C07268=1082.285,311.899,-88.847,175.955,25.912,154.344
C07269=1082.279,311.650,-88.815,175.952,25.909,154.344
C07270=1082.273,311.403,-88.784,175.949,25.904,154.343
C07271=1082.267,311.155,-88.752,175.946,25.900,154.343
C07272=1082.262,310.908,-88.720,175.943,25.896,154.342
C07273=1082.256,310.659,-88.688,175.941,25.892,154.341
C07274=1082.249,310.411,-88.657,175.937,25.888,154.341
C07275=1082.244,310.164,-88.625,175.935,25.884,154.340
C07276=1082.238,309.916,-88.593,175.931,25.880,154.340
C07277=1082.231,309.668,-88.562,175.928,25.876,154.339
C07278=1082.226,309.420,-88.531,175.925,25.872,154.339
C07279=1082.220,309.172,-88.499,175.922,25.868,154.338
C07280=1082.214,308.924,-88.467,175.919,25.864,154.338
C07281=1082.208,308.676,-88.435,175.916,25.860,154.337
C07282=1082.202,308.429,-88.404,175.913,25.856,154.336
C07283=1082.196,308.180,-88.372,175.911,25.852,154.336
C07284=1082.190,307.932,-88.341,175.908,25.848,154.335
C07285=1082.185,307.684,-88.309,175.905,25.844,154.335
C07286=1082.179,307.437,-88.278,175.902,25.840,154.334
C07287=1082.172,307.189,-88.246,175.899,25.836,154.334
C07288=1082.167,306.941,-88.215,175.896,25.832,154.333
C07289=1082.161,306.693,-88.183,175.893,25.828,154.332
C07290=1082.155,306.445,-88.152,175.890,25.824,154.332
C07291=1082.150,306.197,-88.121,175.887,25.820,154.331
C07292=1082.144,305.949,-88.089,175.885,25.816,154.331
C07293=1082.138,305.702,-88.058,175.882,25.812,154.330
C07294=1082.132,305.453,-88.027,175.879,25.808,154.330
C07295=1082.126,305.206,-87.996,175.876,25.804,154.329
C07296=1082.121,304.958,-87.964,175.873,25.800,154.328
C07297=1082.115,304.709,-87.933,175.870,25.796,154.328
C07298=1082.109,304.462,-87.902,175.867,25.792,154.327
C07299=1082.103,304.213,-87.870,175.863,25.788,154.327
C07300=1082.093,303.800,-87.818,175.859,25.781,154.326
C07301=1082.084,303.388,-87.767,175.855,25.775,154.325
C07302=1082.075,302.974,-87.714,175.849,25.768,154.324
C07303=1082.065,302.561,-87.662,175.845,25.762,154.323
C07304=1082.059,302.314,-87.632,175.842,25.758,154.323
C07305=1082.053,302.065,-87.600,175.839,25.753,154.322
C07306=1082.047,301.818,-87.570,175.836,25.749,154.321
C07307=1082.042,301.570,-87.538,175.833,25.746,154.321
C07308=1082.037,301.322,-87.507,175.831,25.742,154.320
C07309=1082.031,301.073,-87.476,175.828,25.738,154.320
C07310=1082.025,300.826,-87.445,175.825,25.734,154.319
C07311=1082.019,300.578,-87.414,175.822,25.730,154.319
C07312=1082.014,300.330,-87.383,175.818,25.726,154.318
C07313=1082.008,300.082,-87.352,175.815,25.722,154.318
C07314=1082.002,299.834,-87.321,175.813,25.718,154.317
C07315=1081.997,299.586,-87.291,175.810,25.714,154.317
C07316=1081.991,299.339,-87.259,175.807,25.710,154.316
C07317=1081.985,299.090,-87.228,175.804,25.706,154.315
C07318=1081.980,298.842,-87.197,175.801,25.702,154.315
C07319=1081.974,298.594,-87.167,175.798,25.698,154.314
C07320=1081.969,298.346,-87.136,175.796,25.695,154.314
C07321=1081.963,298.099,-87.105,175.793,25.690,154.313
C07322=1081.957,297.850,-87.074,175.790,25.686,154.313
C07323=1081.951,297.602,-87.043,175.787,25.682,154.312
C07324=1081.945,297.354,-87.013,175.784,25.678,154.312
C07325=1081.940,297.106,-86.983,175.782,25.675,154.311
C07326=1081.934,296.858,-86.951,175.779,25.671,154.310
C07327=1081.928,296.610,-86.921,175.776,25.667,154.310
C07328=1081.922,296.362,-86.891,175.773,25.663,154.309
C07329=1081.916,296.114,-86.860,175.771,25.660,154.309
C07330=1081.910,295.866,-86.828,175.767,25.656,154.308
C07331=1081.905,295.618,-86.798,175.764,25.652,154.308
C07332=1081.899,295.370,-86.768,175.761,25.648,154.307
C07333=1081.893,295.122,-86.737,175.758,25.644,154.307
C07334=1081.887,294.875,-86.707,175.756,25.641,154.306
C07335=1081.881,294.625,-86.677,175.753,25.637,154.306
C07336=1081.875,294.378,-86.647,175.750,25.633,154.305
C07337=1081.870,294.130,-86.616,175.747,25.629,154.305
C07338=1081.864,293.882,-86.585,175.744,25.625,154.304
C07339=1081.859,293.634,-86.555,175.742,25.621,154.304
C07340=1081.853,293.386,-86.525,175.739,25.618,154.303
C07341=1081.846,293.138,-86.494,175.736,25.614,154.303
C07342=1081.841,292.890,-86.463,175.733,25.610,154.302
C07343=1081.835,292.642,-86.433,175.730,25.607,154.302
C07344=1081.829,292.393,-86.403,175.727,25.603,154.301
C07345=1081.824,292.145,-86.373,175.724,25.599,154.301
C07346=1081.818,291.897,-86.342,175.721,25.595,154.300
C07347=1081.812,291.650,-86.312,175.719,25.591,154.300
C07348=1081.806,291.401,-86.281,175.716,25.588,154.299
C07349=1081.801,291.153,-86.251,175.713,25.584,154.299
C07350=1081.795,290.905,-86.221,175.710,25.580,154.298
C07351=1081.789,290.657,-86.191,175.708,25.576,154.298
C07352=1081.780,290.258,-86.142,175.703,25.570,154.297
C07353=1081.771,289.859,-86.094,175.699,25.564,154.296
C07354=1081.761,289.460,-86.045,175.694,25.558,154.295
C07355=1081.751,289.062,-85.997,175.690,25.552,154.294
C07356=1081.746,288.813,-85.968,175.687,25.548,154.294
C07357=1081.740,288.565,-85.937,175.684,25.545,154.294
C07358=1081.734,288.318,-85.907,175.681,25.541,154.293
C07359=1081.729,288.069,-85.877,175.679,25.537,154.292
C07360=1081.723,287.821,-85.847,175.675,25.533,154.292
C07361=1081.717,287.573,-85.818,175.672,25.530,154.292
C07362=1081.711,287.325,-85.788,175.670,25.526,154.291
C07363=1081.705,287.077,-85.758,175.667,25.522,154.290
C07364=1081.699,286.829,-85.728,175.664,25.519,154.290
C07365=1081.694,286.581,-85.698,175.661,25.515,154.290
C07366=1081.688,286.333,-85.668,175.659,25.511,154.289
C07367=1081.682,286.085,-85.638,175.656,25.507,154.288
C07368=1081.676,285.837,-85.608,175.653,25.504,154.288
C07369=1081.670,285.589,-85.579,175.651,25.500,154.288
C07370=1081.665,285.340,-85.549,175.648,25.496,154.287
C07371=1081.659,285.092,-85.519,175.644,25.493,154.287
C07372=1081.653,284.844,-85.489,175.641,25.489,154.286
C07373=1081.647,284.596,-85.460,175.639,25.485,154.286
C07374=1081.642,284.348,-85.429,175.636,25.482,154.285
C07375=1081.636,284.099,-85.400,175.633,25.478,154.285
C07376=1081.631,283.851,-85.370,175.631,25.474,154.284
C07377=1081.624,283.603,-85.340,175.628,25.471,154.284
C07378=1081.618,283.355,-85.311,175.625,25.467,154.283
C07379=1081.613,283.107,-85.281,175.623,25.463,154.283
C07380=1081.607,282.859,-85.251,175.620,25.460,154.282
C07381=1081.601,282.611,-85.222,175.617,25.456,154.282
C07382=1081.595,282.362,-85.192,175.614,25.452,154.281
C07383=1081.590,282.114,-85.163,175.611,25.449,154.281
C07384=1081.584,281.865,-85.133,175.608,25.445,154.280
C07385=1081.578,281.619,-85.104,175.606,25.441,154.280
C07386=1081.573,281.370,-85.074,175.603,25.438,154.279
C07387=1081.567,281.122,-85.044,175.600,25.434,154.279
C07388=1081.561,280.873,-85.015,175.598,25.430,154.278
C07389=1081.556,280.625,-84.986,175.595,25.427,154.278
C07390=1081.550,280.377,-84.956,175.592,25.423,154.277
C07391=1081.544,280.128,-84.927,175.590,25.419,154.277
C07392=1081.538,279.881,-84.897,175.587,25.416,154.276
C07393=1081.532,279.633,-84.868,175.584,25.412,154.276
C07394=1081.526,279.384,-84.838,175.581,25.408,154.275
C07395=1081.521,279.137,-84.809,175.578,25.405,154.275
C07396=1081.515,278.888,-84.780,175.575,25.401,154.274
C07397=1081.509,278.640,-84.751,175.573,25.398,154.274
C07398=1081.503,278.392,-84.721,175.570,25.394,154.274
C07399=1081.498,278.143,-84.691,175.567,25.390,154.273
C07400=1081.492,277.895,-84.662,175.565,25.387,154.273
C07401=1081.486,277.647,-84.633,175.562,25.383,154.272
C07402=1081.481,277.399,-84.605,175.559,25.379,154.272
C07403=1081.475,277.150,-84.575,175.557,25.376,154.271
C07404=1081.466,276.762,-84.529,175.552,25.370,154.270
C07405=1081.457,276.373,-84.484,175.547,25.364,154.270
C07406=1081.448,275.983,-84.438,175.544,25.359,154.269
C07407=1081.438,275.594,-84.392,175.539,25.353,154.268
C07408=1081.434,275.346,-84.363,175.536,25.349,154.268
C07409=1081.427,275.097,-84.334,175.534,25.346,154.267
C07410=1081.421,274.849,-84.305,175.531,25.342,154.267
C07411=1081.416,274.601,-84.275,175.528,25.339,154.266
C07412=1081.410,274.353,-84.247,175.526,25.335,154.266
C07413=1081.405,274.104,-84.218,175.523,25.331,154.265
C07414=1081.399,273.856,-84.189,175.520,25.328,154.265
C07415=1081.392,273.608,-84.160,175.517,25.324,154.264
C07416=1081.388,273.360,-84.131,175.514,25.321,154.264
C07417=1081.381,273.112,-84.102,175.512,25.317,154.264
C07418=1081.375,272.863,-84.073,175.509,25.314,154.263
C07419=1081.370,272.614,-84.044,175.507,25.311,154.263
C07420=1081.364,272.367,-84.016,175.504,25.307,154.262
C07421=1081.358,272.119,-83.987,175.501,25.303,154.262
C07422=1081.352,271.870,-83.958,175.499,25.300,154.261
C07423=1081.347,271.622,-83.929,175.496,25.296,154.261
C07424=1081.341,271.374,-83.900,175.493,25.292,154.260
C07425=1081.335,271.125,-83.872,175.490,25.289,154.260
C07426=1081.329,270.877,-83.843,175.487,25.285,154.259
C07427=1081.324,270.629,-83.814,175.485,25.282,154.259
C07428=1081.318,270.381,-83.785,175.482,25.278,154.259
C07429=1081.312,270.132,-83.757,175.480,25.275,154.258
C07430=1081.306,269.885,-83.728,175.477,25.271,154.258
C07431=1081.301,269.636,-83.699,175.474,25.267,154.257
C07432=1081.295,269.387,-83.670,175.472,25.264,154.257
C07433=1081.290,269.139,-83.642,175.469,25.260,154.256
C07434=1081.283,268.891,-83.613,175.466,25.257,154.256
C07435=1081.277,268.643,-83.585,175.463,25.253,154.255
C07436=1081.272,268.394,-83.557,175.460,25.250,154.255
C07437=1081.266,268.146,-83.528,175.458,25.247,154.255
C07438=1081.261,267.897,-83.499,175.455,25.243,154.254
C07439=1081.255,267.650,-83.470,175.453,25.240,154.254
C07440=1081.249,267.401,-83.442,175.450,25.236,154.253
C07441=1081.243,267.152,-83.413,175.448,25.232,154.253
C07442=1081.237,266.905,-83.385,175.445,25.229,154.252
C07443=1081.231,266.656,-83.356,175.442,25.225,154.252
C07444=1081.226,266.408,-83.328,175.439,25.222,154.251
C07445=1081.220,266.160,-83.299,175.436,25.218,154.251
C07446=1081.214,265.911,-83.271,175.434,25.215,154.250
C07447=1081.209,265.663,-83.243,175.431,25.211,154.250
C07448=1081.203,265.414,-83.215,175.429,25.208,154.250
C07449=1081.198,265.167,-83.186,175.426,25.204,154.249
C07450=1081.192,264.918,-83.157,175.424,25.201,154.249
C07451=1081.186,264.670,-83.129,175.421,25.197,154.248
C07452=1081.180,264.421,-83.101,175.418,25.193,154.248
C07453=1081.175,264.173,-83.073,175.415,25.190,154.247
C07454=1081.169,263.924,-83.045,175.412,25.186,154.247
C07455=1081.162,263.677,-83.016,175.410,25.183,154.246
C07456=1081.154,263.290,-82.973,175.406,25.178,154.246
C07457=1081.145,262.904,-82.929,175.402,25.172,154.245
C07458=1081.135,262.518,-82.885,175.397,25.167,154.244
C07459=1081.126,262.132,-82.841,175.394,25.162,154.244
C07460=1081.120,261.883,-82.813,175.390,25.158,154.243
C07461=1081.115,261.635,-82.785,175.388,25.155,154.243
C07462=1081.108,261.387,-82.757,175.385,25.151,154.242
C07463=1081.103,261.139,-82.729,175.383,25.148,154.242
C07464=1081.097,260.890,-82.701,175.380,25.144,154.242
C07465=1081.092,260.642,-82.673,175.378,25.141,154.241
C07466=1081.085,260.393,-82.645,175.375,25.137,154.241
C07467=1081.079,260.145,-82.617,175.372,25.134,154.240
C07468=1081.074,259.897,-82.589,175.370,25.131,154.240
C07469=1081.068,259.649,-82.561,175.366,25.127,154.240
C07470=1081.062,259.400,-82.533,175.364,25.124,154.239
C07471=1081.056,259.152,-82.506,175.361,25.120,154.239
C07472=1081.051,258.903,-82.478,175.359,25.117,154.238
C07473=1081.045,258.655,-82.450,175.356,25.113,154.238
C07474=1081.039,258.406,-82.422,175.354,25.110,154.237
C07475=1081.033,258.158,-82.394,175.351,25.106,154.237
C07476=1081.027,257.909,-82.366,175.349,25.103,154.236
C07477=1081.021,257.662,-82.339,175.346,25.099,154.236
C07478=1081.016,257.412,-82.311,175.343,25.096,154.236
C07479=1081.010,257.164,-82.283,175.340,25.093,154.235
C07480=1081.004,256.916,-82.255,175.338,25.089,154.235
C07481=1080.998,256.668,-82.227,175.335,25.085,154.234
C07482=1080.993,256.419,-82.200,175.333,25.082,154.234
C07483=1080.986,256.171,-82.172,175.330,25.079,154.233
C07484=1080.981,255.923,-82.144,175.328,25.075,154.233
C07485=1080.975,255.674,-82.116,175.325,25.072,154.233
C07486=1080.969,255.426,-82.089,175.322,25.068,154.232
C07487=1080.964,255.178,-82.061,175.319,25.065,154.232
C07488=1080.958,254.929,-82.033,175.317,25.061,154.231
C07489=1080.952,254.680,-82.006,175.314,25.058,154.231
C07490=1080.946,254.432,-81.978,175.312,25.055,154.230
C07491=1080.941,254.183,-81.951,175.309,25.051,154.230
C07492=1080.935,253.935,-81.923,175.307,25.048,154.229
C07493=1080.929,253.686,-81.895,175.304,25.044,154.229
C07494=1080.924,253.438,-81.868,175.302,25.041,154.229
C07495=1080.918,253.190,-81.841,175.299,25.037,154.228
C07496=1080.913,252.941,-81.813,175.296,25.034,154.228
C07497=1080.906,252.693,-81.786,175.294,25.031,154.227
C07498=1080.901,252.444,-81.758,175.291,25.027,154.227
C07499=1080.896,252.196,-81.730,175.289,25.023,154.226
C07500=1080.890,251.947,-81.703,175.286,25.020,154.226
C07501=1080.884,251.699,-81.675,175.284,25.016,154.226
C07502=1080.879,251.451,-81.649,175.281,25.013,154.225
C07503=1080.873,251.202,-81.620,175.279,25.010,154.225
C07504=1080.868,250.953,-81.593,175.276,25.006,154.224
C07505=1080.862,250.706,-81.566,175.273,25.003,154.224
C07506=1080.857,250.457,-81.539,175.270,24.999,154.223
C07507=1080.850,250.208,-81.511,175.268,24.995,154.223
C07508=1080.842,249.820,-81.468,175.265,24.990,154.222
C07509=1080.833,249.431,-81.426,175.260,24.985,154.222
C07510=1080.824,249.042,-81.383,175.256,24.979,154.221
C07511=1080.815,248.654,-81.340,175.252,24.974,154.220
C07512=1080.810,248.404,-81.313,175.250,24.970,154.220
C07513=1080.804,248.156,-81.286,175.247,24.966,154.219
C07514=1080.799,247.908,-81.258,175.245,24.963,154.219
C07515=1080.793,247.659,-81.231,175.242,24.960,154.218
C07516=1080.788,247.411,-81.204,175.239,24.956,154.218
C07517=1080.782,247.162,-81.177,175.237,24.953,154.217
C07518=1080.776,246.914,-81.149,175.234,24.949,154.217
C07519=1080.770,246.665,-81.122,175.232,24.946,154.217
C07520=1080.765,246.417,-81.096,175.229,24.942,154.216
C07521=1080.759,246.168,-81.069,175.227,24.939,154.216
C07522=1080.754,245.920,-81.042,175.225,24.936,154.215
C07523=1080.747,245.671,-81.015,175.222,24.932,154.215
C07524=1080.742,245.423,-80.987,175.220,24.929,154.214
C07525=1080.736,245.174,-80.960,175.217,24.925,154.214
C07526=1080.730,244.926,-80.934,175.214,24.922,154.214
C07527=1080.725,244.677,-80.906,175.211,24.918,154.213
C07528=1080.720,244.429,-80.880,175.209,24.915,154.213
C07529=1080.713,244.180,-80.853,175.207,24.912,154.212
C07530=1080.707,243.932,-80.826,175.204,24.908,154.212
C07531=1080.702,243.683,-80.799,175.202,24.905,154.211
C07532=1080.697,243.435,-80.772,175.199,24.901,154.211
C07533=1080.691,243.186,-80.746,175.197,24.898,154.211
C07534=1080.686,242.937,-80.718,175.194,24.895,154.210
C07535=1080.680,242.689,-80.692,175.192,24.891,154.210
C07536=1080.674,242.441,-80.665,175.189,24.888,154.209
C07537=1080.668,242.192,-80.638,175.186,24.884,154.209
C07538=1080.662,241.943,-80.611,175.184,24.881,154.209
C07539=1080.656,241.695,-80.585,175.182,24.878,154.208
C07540=1080.651,241.447,-80.558,175.179,24.874,154.208
C07541=1080.645,241.198,-80.531,175.177,24.871,154.207
C07542=1080.640,240.950,-80.504,175.174,24.867,154.207
C07543=1080.634,240.701,-80.478,175.172,24.864,154.206
C07544=1080.628,240.453,-80.451,175.169,24.861,154.206
C07545=1080.622,240.204,-80.424,175.166,24.857,154.206
C07546=1080.616,239.955,-80.398,175.164,24.853,154.205
C07547=1080.611,239.706,-80.371,175.161,24.850,154.205
C07548=1080.605,239.458,-80.345,175.159,24.847,154.204
C07549=1080.599,239.210,-80.318,175.157,24.844,154.204
C07550=1080.593,238.961,-80.291,175.154,24.840,154.204
C07551=1080.588,238.712,-80.265,175.152,24.836,154.203
C07552=1080.582,238.464,-80.239,175.150,24.833,154.203
C07553=1080.576,238.216,-80.212,175.146,24.830,154.202
C07554=1080.571,237.967,-80.185,175.144,24.827,154.202
C07555=1080.565,237.719,-80.159,175.141,24.823,154.201
C07556=1080.559,237.470,-80.133,175.139,24.820,154.201
C07557=1080.554,237.222,-80.106,175.137,24.816,154.200
C07558=1080.548,236.973,-80.080,175.134,24.813,154.200
C07559=1080.542,236.724,-80.054,175.132,24.810,154.200
C07560=1080.533,236.329,-80.011,175.128,24.804,154.199
C07561=1080.524,235.934,-79.969,175.124,24.799,154.198
C07562=1080.515,235.538,-79.927,175.120,24.793,154.198
C07563=1080.506,235.142,-79.885,175.116,24.788,154.197
C07564=1080.500,234.893,-79.859,175.113,24.784,154.197
C07565=1080.495,234.645,-79.832,175.111,24.781,154.196
C07566=1080.489,234.396,-79.806,175.108,24.777,154.196
C07567=1080.483,234.147,-79.780,175.106,24.774,154.195
C07568=1080.478,233.899,-79.754,175.104,24.771,154.195
C07569=1080.472,233.651,-79.728,175.101,24.767,154.194
C07570=1080.466,233.402,-79.702,175.099,24.764,154.194
C07571=1080.461,233.154,-79.676,175.097,24.760,154.194
C07572=1080.455,232.905,-79.650,175.094,24.757,154.193
C07573=1080.449,232.656,-79.623,175.092,24.754,154.193
C07574=1080.444,232.407,-79.597,175.089,24.751,154.192
C07575=1080.438,232.159,-79.570,175.086,24.747,154.192
C07576=1080.432,231.910,-79.545,175.084,24.743,154.191
C07577=1080.426,231.662,-79.518,175.082,24.740,154.191
C07578=1080.421,231.413,-79.492,175.079,24.737,154.191
C07579=1080.415,231.164,-79.467,175.077,24.734,154.190
C07580=1080.410,230.916,-79.440,175.075,24.730,154.190
C07581=1080.404,230.668,-79.415,175.072,24.726,154.189
C07582=1080.398,230.419,-79.388,175.070,24.723,154.189
C07583=1080.393,230.170,-79.362,175.067,24.720,154.188
C07584=1080.387,229.921,-79.336,175.064,24.716,154.188
C07585=1080.381,229.673,-79.310,175.062,24.713,154.188
C07586=1080.375,229.424,-79.284,175.060,24.710,154.187
C07587=1080.369,229.176,-79.259,175.057,24.706,154.187
C07588=1080.364,228.927,-79.233,175.055,24.703,154.186
C07589=1080.358,228.678,-79.207,175.053,24.700,154.186
C07590=1080.352,228.430,-79.182,175.051,24.696,154.186
C07591=1080.347,228.181,-79.156,175.048,24.693,154.185
C07592=1080.341,227.932,-79.130,175.045,24.690,154.185
C07593=1080.335,227.684,-79.104,175.043,24.687,154.184
C07594=1080.329,227.435,-79.078,175.040,24.683,154.184
C07595=1080.323,227.187,-79.052,175.038,24.679,154.183
C07596=1080.318,226.938,-79.027,175.036,24.676,154.183
C07597=1080.313,226.689,-79.001,175.033,24.673,154.183
C07598=1080.307,226.441,-78.976,175.031,24.669,154.182
C07599=1080.301,226.192,-78.949,175.029,24.666,154.182
C07600=1080.295,225.944,-78.924,175.027,24.663,154.181
C07601=1080.289,225.695,-78.898,175.024,24.659,154.181
C07602=1080.283,225.447,-78.873,175.022,24.656,154.181
C07603=1080.278,225.198,-78.847,175.019,24.653,154.180
C07604=1080.273,224.949,-78.821,175.016,24.649,154.180
C07605=1080.266,224.700,-78.795,175.014,24.645,154.179
C07606=1080.261,224.452,-78.770,175.012,24.642,154.179
C07607=1080.255,224.203,-78.745,175.010,24.639,154.178
C07608=1080.250,223.954,-78.719,175.007,24.636,154.178
C07609=1080.244,223.705,-78.693,175.005,24.632,154.178
C07610=1080.239,223.457,-78.668,175.003,24.629,154.177
C07611=1080.232,223.208,-78.642,175.000,24.625,154.177
C07612=1080.224,222.805,-78.601,174.996,24.620,154.176
C07613=1080.214,222.400,-78.559,174.993,24.614,154.175
C07614=1080.205,221.996,-78.517,174.988,24.609,154.175
C07615=1080.196,221.592,-78.476,174.985,24.603,154.174
C07616=1080.190,221.343,-78.450,174.982,24.600,154.174
C07617=1080.184,221.095,-78.425,174.980,24.597,154.173
C07618=1080.179,220.847,-78.400,174.977,24.593,154.173
C07619=1080.173,220.597,-78.375,174.975,24.590,154.172
C07620=1080.167,220.349,-78.349,174.973,24.587,154.172
C07621=1080.161,220.100,-78.324,174.971,24.583,154.172
C07622=1080.155,219.852,-78.299,174.968,24.580,154.171
C07623=1080.150,219.603,-78.273,174.966,24.577,154.171
C07624=1080.144,219.354,-78.248,174.964,24.573,154.170
C07625=1080.139,219.106,-78.224,174.962,24.570,154.170
C07626=1080.133,218.857,-78.198,174.959,24.566,154.169
C07627=1080.127,218.608,-78.172,174.956,24.563,154.169
C07628=1080.121,218.360,-78.147,174.954,24.560,154.169
C07629=1080.116,218.110,-78.122,174.952,24.557,154.168
C07630=1080.110,217.862,-78.097,174.949,24.553,154.168
C07631=1080.104,217.614,-78.072,174.947,24.549,154.167
C07632=1080.098,217.365,-78.047,174.945,24.546,154.167
C07633=1080.093,217.116,-78.021,174.943,24.543,154.166
C07634=1080.087,216.868,-77.996,174.940,24.539,154.166
C07635=1080.081,216.618,-77.972,174.938,24.536,154.166
C07636=1080.076,216.370,-77.947,174.936,24.533,154.165
C07637=1080.070,216.121,-77.921,174.934,24.529,154.165
C07638=1080.064,215.872,-77.896,174.930,24.526,154.164
C07639=1080.059,215.624,-77.871,174.928,24.523,154.164
C07640=1080.053,215.375,-77.846,174.926,24.519,154.164
C07641=1080.048,215.127,-77.821,174.924,24.516,154.163
C07642=1080.042,214.878,-77.796,174.921,24.512,154.163
C07643=1080.037,214.629,-77.771,174.919,24.509,154.162
C07644=1080.030,214.381,-77.746,174.917,24.506,154.162
C07645=1080.024,214.131,-77.721,174.915,24.503,154.161
C07646=1080.020,213.883,-77.696,174.913,24.499,154.161
C07647=1080.013,213.634,-77.671,174.910,24.495,154.161
C07648=1080.008,213.386,-77.646,174.908,24.492,154.160
C07649=1080.002,213.137,-77.621,174.905,24.489,154.160
C07650=1079.997,212.889,-77.597,174.903,24.486,154.159
C07651=1079.991,212.639,-77.572,174.900,24.482,154.159
C07652=1079.986,212.391,-77.547,174.898,24.478,154.158
C07653=1079.980,212.142,-77.522,174.896,24.475,154.158
C07654=1079.974,211.894,-77.497,174.894,24.472,154.158
C07655=1079.968,211.644,-77.472,174.892,24.469,154.157
C07656=1079.963,211.396,-77.447,174.889,24.465,154.157
C07657=1079.957,211.147,-77.423,174.887,24.461,154.156
C07658=1079.952,210.899,-77.398,174.885,24.458,154.156
C07659=1079.945,210.650,-77.373,174.883,24.455,154.156
C07660=1079.940,210.401,-77.349,174.881,24.452,154.155
C07661=1079.934,210.152,-77.324,174.877,24.448,154.155
C07662=1079.929,209.904,-77.299,174.875,24.445,154.154
C07663=1079.923,209.655,-77.275,174.873,24.441,154.154
C07664=1079.913,209.254,-77.235,174.870,24.436,154.153
C07665=1079.905,208.855,-77.196,174.866,24.431,154.153
C07666=1079.895,208.455,-77.156,174.863,24.425,154.152
C07667=1079.886,208.055,-77.116,174.859,24.420,154.151
C07668=1079.863,207.021,-77.017,174.758,24.366,154.153
C07669=1079.856,206.772,-76.993,174.755,24.364,154.153
C07670=1079.851,206.523,-76.969,174.753,24.361,154.152
C07671=1079.846,206.275,-76.944,174.750,24.359,154.152
C07672=1079.841,206.026,-76.920,174.748,24.357,154.152
C07673=1079.834,205.776,-76.897,174.746,24.354,154.152
C07674=1079.829,205.528,-76.872,174.743,24.352,154.152
C07675=1079.824,205.279,-76.848,174.740,24.349,154.151
C07676=1079.818,205.031,-76.825,174.738,24.347,154.151
C07677=1079.813,204.782,-76.801,174.735,24.344,154.151
C07678=1079.807,204.532,-76.776,174.733,24.342,154.151
C07679=1079.801,204.284,-76.753,174.731,24.339,154.151
C07680=1079.796,204.035,-76.729,174.728,24.337,154.150
C07681=1079.790,203.787,-76.706,174.726,24.334,154.150
C07682=1079.784,203.538,-76.681,174.724,24.332,154.150
C07683=1079.779,203.289,-76.658,174.721,24.329,154.150
C07684=1079.773,203.040,-76.634,174.719,24.327,154.150
C07685=1079.767,202.791,-76.609,174.717,24.325,154.149
C07686=1079.762,202.542,-76.586,174.714,24.322,154.149
C07687=1079.756,202.294,-76.562,174.712,24.320,154.149
C07688=1079.750,202.046,-76.539,174.710,24.318,154.149
C07689=1079.745,201.796,-76.515,174.707,24.315,154.149
C07690=1079.739,201.547,-76.491,174.705,24.313,154.148
C07691=1079.734,201.298,-76.467,174.702,24.310,154.148
C07692=1079.728,201.050,-76.444,174.700,24.308,154.148
C07693=1079.722,200.801,-76.421,174.698,24.306,154.148
C07694=1079.717,200.552,-76.397,174.695,24.303,154.148
C07695=1079.710,200.303,-76.373,174.693,24.301,154.147
C07696=1079.705,200.054,-76.349,174.690,24.299,154.147
C07697=1079.699,199.805,-76.326,174.688,24.296,154.147
C07698=1079.693,199.557,-76.302,174.686,24.294,154.147
C07699=1079.688,199.308,-76.279,174.683,24.292,154.147
C07700=1079.682,199.060,-76.255,174.681,24.289,154.146
C07701=1079.677,198.810,-76.232,174.679,24.287,154.146
C07702=1079.671,198.561,-76.208,174.676,24.285,154.146
C07703=1079.665,198.313,-76.185,174.674,24.282,154.146
C07704=1079.660,198.063,-76.161,174.672,24.280,154.146
C07705=1079.654,197.815,-76.138,174.669,24.278,154.146
C07706=1079.648,197.566,-76.115,174.667,24.275,154.145
C07707=1079.643,197.318,-76.090,174.664,24.273,154.145
C07708=1079.637,197.069,-76.067,174.662,24.271,154.145
C07709=1079.631,196.820,-76.044,174.660,24.268,154.145
C07710=1079.626,196.571,-76.020,174.657,24.266,154.145
C07711=1079.620,196.322,-75.997,174.655,24.264,154.145
C07712=1079.615,196.073,-75.974,174.653,24.261,154.144
C07713=1079.609,195.824,-75.950,174.650,24.259,154.144
C07714=1079.603,195.575,-75.927,174.648,24.256,154.144
C07715=1079.597,195.326,-75.904,174.646,24.255,154.144
C07716=1079.592,195.078,-75.879,174.644,24.252,154.144
C07717=1079.586,194.829,-75.857,174.642,24.250,154.143
C07718=1079.580,194.580,-75.834,174.639,24.247,154.143
C07719=1079.575,194.331,-75.811,174.637,24.245,154.143
C07720=1079.569,194.082,-75.786,174.635,24.243,154.143
C07721=1079.564,193.834,-75.763,174.632,24.240,154.143
C07722=1079.558,193.585,-75.741,174.630,24.238,154.142
C07723=1079.553,193.335,-75.717,174.628,24.236,154.142
C07724=1079.547,193.087,-75.694,174.625,24.233,154.142
C07725=1079.541,192.838,-75.670,174.623,24.231,154.142
C07726=1079.535,192.589,-75.647,174.620,24.229,154.142
C07727=1079.530,192.340,-75.624,174.618,24.226,154.141
C07728=1079.525,192.091,-75.601,174.616,24.224,154.141
C07729=1079.519,191.812,-75.575,174.614,24.221,154.141
C07730=1079.512,191.532,-75.549,174.611,24.218,154.141
C07731=1079.506,191.252,-75.523,174.608,24.216,154.141
C07732=1079.500,190.972,-75.497,174.606,24.213,154.140
C07733=1079.494,190.723,-75.474,174.603,24.211,154.140
C07734=1079.489,190.475,-75.451,174.601,24.208,154.140
C07735=1079.484,190.226,-75.427,174.599,24.206,154.140
C07736=1079.478,189.977,-75.405,174.596,24.203,154.139
C07737=1079.472,189.728,-75.382,174.595,24.201,154.139
C07738=1079.467,189.479,-75.359,174.593,24.199,154.139
C07739=1079.462,189.230,-75.335,174.590,24.197,154.139
C07740=1079.456,188.981,-75.312,174.588,24.194,154.139
C07741=1079.450,188.732,-75.289,174.585,24.192,154.138
C07742=1079.444,188.483,-75.266,174.583,24.189,154.138
C07743=1079.439,188.235,-75.244,174.581,24.187,154.138
C07744=1079.434,187.986,-75.220,174.578,24.185,154.138
C07745=1079.429,187.737,-75.197,174.576,24.182,154.138
C07746=1079.423,187.488,-75.174,174.574,24.180,154.137
C07747=1079.417,187.239,-75.151,174.572,24.177,154.137
C07748=1079.411,186.990,-75.128,174.570,24.175,154.137
C07749=1079.406,186.741,-75.105,174.568,24.172,154.137
C07750=1079.401,186.493,-75.082,174.565,24.170,154.137
C07751=1079.396,186.244,-75.059,174.563,24.168,154.136
C07752=1079.390,185.995,-75.036,174.561,24.165,154.136
C07753=1079.384,185.746,-75.013,174.558,24.163,154.136
C07754=1079.379,185.496,-74.991,174.556,24.161,154.136
C07755=1079.374,185.248,-74.969,174.554,24.159,154.136
C07756=1079.369,184.999,-74.945,174.552,24.156,154.135
C07757=1079.362,184.750,-74.923,174.550,24.154,154.135
C07758=1079.356,184.502,-74.900,174.547,24.152,154.135
C07759=1079.351,184.253,-74.877,174.545,24.149,154.135
C07760=1079.345,184.003,-74.855,174.543,24.147,154.135
C07761=1079.339,183.754,-74.832,174.540,24.145,154.135
C07762=1079.333,183.506,-74.809,174.538,24.142,154.134
C07763=1079.327,183.257,-74.786,174.536,24.140,154.134
C07764=1079.322,183.007,-74.764,174.534,24.138,154.134
C07765=1079.317,182.759,-74.742,174.532,24.136,154.134
C07766=1079.310,182.510,-74.719,174.529,24.133,154.134
C07767=1079.305,182.262,-74.696,174.527,24.131,154.133
C07768=1079.299,182.012,-74.674,174.525,24.129,154.133
C07769=1079.293,181.763,-74.651,174.523,24.127,154.133
C07770=1079.288,181.514,-74.628,174.521,24.125,154.133
C07771=1079.281,181.265,-74.606,174.518,24.122,154.133
C07772=1079.276,181.016,-74.584,174.516,24.120,154.133
C07773=1079.271,180.768,-74.561,174.514,24.118,154.132
C07774=1079.264,180.519,-74.539,174.511,24.115,154.132
C07775=1079.259,180.270,-74.516,174.509,24.113,154.132
C07776=1079.253,180.021,-74.493,174.507,24.111,154.132
C07777=1079.248,179.771,-74.471,174.505,24.109,154.132
C07778=1079.241,179.523,-74.449,174.503,24.106,154.131
C07779=1079.236,179.274,-74.427,174.500,24.104,154.131
C07780=1079.231,179.025,-74.404,174.498,24.102,154.131
C07781=1079.225,178.776,-74.381,174.497,24.099,154.131
C07782=1079.219,178.527,-74.359,174.494,24.097,154.131
C07783=1079.214,178.279,-74.337,174.492,24.095,154.131
C07784=1079.208,178.029,-74.315,174.489,24.093,154.130
C07785=1079.202,177.781,-74.292,174.487,24.090,154.130
C07786=1079.196,177.531,-74.270,174.485,24.088,154.130
C07787=1079.190,177.282,-74.247,174.483,24.086,154.130
C07788=1079.185,177.034,-74.226,174.481,24.083,154.130
C07789=1079.179,176.785,-74.203,174.479,24.081,154.129
C07790=1079.174,176.535,-74.181,174.476,24.079,154.129
C07791=1079.167,176.287,-74.158,174.474,24.076,154.129
C07792=1079.162,176.038,-74.136,174.472,24.074,154.129
C07793=1079.156,175.757,-74.111,174.469,24.071,154.129
C07794=1079.149,175.478,-74.087,174.467,24.069,154.129
C07795=1079.143,175.197,-74.061,174.465,24.066,154.128
C07796=1079.137,174.917,-74.036,174.462,24.064,154.128
C07797=1079.131,174.668,-74.014,174.460,24.061,154.128
C07798=1079.126,174.419,-73.992,174.458,24.059,154.128
C07799=1079.120,174.170,-73.970,174.456,24.057,154.127
C07800=1079.114,173.921,-73.947,174.454,24.055,154.127
C07801=1079.109,173.672,-73.925,174.452,24.052,154.127
C07802=1079.103,173.424,-73.903,174.449,24.050,154.127
C07803=1079.097,173.174,-73.881,174.447,24.048,154.127
C07804=1079.092,172.926,-73.859,174.445,24.045,154.126
C07805=1079.086,172.677,-73.837,174.443,24.043,154.126
C07806=1079.081,172.427,-73.814,174.441,24.041,154.126
C07807=1079.076,172.179,-73.793,174.438,24.038,154.126
C07808=1079.070,171.929,-73.771,174.437,24.036,154.126
C07809=1079.064,171.680,-73.748,174.435,24.034,154.125
C07810=1079.059,171.432,-73.726,174.432,24.031,154.125
C07811=1079.053,171.182,-73.704,174.430,24.029,154.125
C07812=1079.048,170.934,-73.683,174.428,24.027,154.125
C07813=1079.042,170.685,-73.660,174.426,24.025,154.125
C07814=1079.036,170.436,-73.638,174.424,24.022,154.124
C07815=1079.031,170.187,-73.617,174.421,24.020,154.124
C07816=1079.025,169.938,-73.595,174.419,24.017,154.124
C07817=1079.020,169.689,-73.572,174.418,24.015,154.124
C07818=1079.014,169.440,-73.550,174.415,24.013,154.124
C07819=1079.008,169.191,-73.528,174.413,24.010,154.123
C07820=1079.003,168.942,-73.507,174.411,24.008,154.123
C07821=1078.997,168.693,-73.485,174.409,24.006,154.123
C07822=1078.992,168.444,-73.463,174.407,24.004,154.123
C07823=1078.986,168.195,-73.440,174.405,24.001,154.123
C07824=1078.981,167.946,-73.419,174.403,23.999,154.122
C07825=1078.975,167.697,-73.397,174.401,23.996,154.122
C07826=1078.970,167.448,-73.375,174.398,23.994,154.122
C07827=1078.964,167.199,-73.353,174.396,23.991,154.122
C07828=1078.959,166.950,-73.332,174.395,23.990,154.122
C07829=1078.953,166.701,-73.310,174.392,23.987,154.121
C07830=1078.948,166.452,-73.288,174.390,23.985,154.121
C07831=1078.942,166.203,-73.266,174.388,23.982,154.121
C07832=1078.937,165.954,-73.245,174.386,23.980,154.121
C07833=1078.931,165.705,-73.223,174.384,23.977,154.121
C07834=1078.926,165.456,-73.201,174.382,23.975,154.120
C07835=1078.920,165.207,-73.179,174.379,23.973,154.120
C07836=1078.915,164.958,-73.158,174.378,23.971,154.120
C07837=1078.909,164.709,-73.136,174.376,23.968,154.120
C07838=1078.904,164.460,-73.114,174.373,23.966,154.120
C07839=1078.898,164.211,-73.092,174.372,23.963,154.119
C07840=1078.893,163.962,-73.071,174.370,23.961,154.119
C07841=1078.887,163.713,-73.049,174.367,23.958,154.119
C07842=1078.882,163.464,-73.027,174.365,23.956,154.119
C07843=1078.876,163.215,-73.005,174.364,23.954,154.118
C07844=1078.871,162.966,-72.984,174.361,23.952,154.118
C07845=1078.866,162.718,-72.962,174.359,23.949,154.118
C07846=1078.860,162.468,-72.940,174.357,23.947,154.118
C07847=1078.855,162.220,-72.919,174.355,23.944,154.118
C07848=1078.849,161.970,-72.897,174.353,23.942,154.117
C07849=1078.844,161.721,-72.876,174.351,23.940,154.117
C07850=1078.839,161.472,-72.854,174.349,23.937,154.117
C07851=1078.833,161.223,-72.832,174.347,23.935,154.117
C07852=1078.828,160.974,-72.811,174.344,23.933,154.117
C07853=1078.821,160.725,-72.790,174.343,23.930,154.116
C07854=1078.816,160.477,-72.768,174.341,23.928,154.116
C07855=1078.811,160.227,-72.747,174.338,23.926,154.116
C07856=1078.802,159.890,-72.718,174.336,23.923,154.116
C07857=1078.797,159.632,-72.696,174.334,23.921,154.115
C07858=1078.792,159.373,-72.673,174.332,23.918,154.115
C07859=1078.785,159.114,-72.652,174.329,23.916,154.115
C07860=1078.779,158.856,-72.629,174.328,23.913,154.115
C07861=1078.774,158.607,-72.607,174.325,23.911,154.115
C07862=1078.768,158.357,-72.586,174.323,23.908,154.114
C07863=1078.762,158.109,-72.565,174.322,23.907,154.114
C07864=1078.757,157.860,-72.544,174.319,23.904,154.114
C07865=1078.751,157.610,-72.523,174.317,23.902,154.114
C07866=1078.746,157.362,-72.501,174.316,23.900,154.114
C07867=1078.740,157.112,-72.479,174.313,23.897,154.113
C07868=1078.735,156.863,-72.459,174.311,23.895,154.113
C07869=1078.729,156.615,-72.438,174.310,23.893,154.113
C07870=1078.723,156.366,-72.416,174.307,23.890,154.113
C07871=1078.718,156.116,-72.395,174.305,23.888,154.113
C07872=1078.712,155.867,-72.374,174.303,23.886,154.112
C07873=1078.706,155.619,-72.352,174.301,23.883,154.112
C07874=1078.702,155.369,-72.331,174.299,23.881,154.112
C07875=1078.695,155.120,-72.310,174.297,23.879,154.112
C07876=1078.690,154.871,-72.289,174.295,23.876,154.112
C07877=1078.684,154.622,-72.267,174.293,23.874,154.111
C07878=1078.678,154.373,-72.246,174.291,23.872,154.111
C07879=1078.673,154.124,-72.226,174.289,23.869,154.111
C07880=1078.667,153.875,-72.204,174.287,23.867,154.111
C07881=1078.662,153.626,-72.183,174.285,23.865,154.111
C07882=1078.656,153.377,-72.162,174.283,23.863,154.110
C07883=1078.650,153.128,-72.141,174.281,23.860,154.110
C07884=1078.645,152.879,-72.120,174.279,23.858,154.110
C07885=1078.639,152.630,-72.099,174.277,23.855,154.110
C07886=1078.633,152.381,-72.078,174.275,23.853,154.110
C07887=1078.628,152.132,-72.057,174.273,23.851,154.109
C07888=1078.622,151.883,-72.036,174.271,23.849,154.109
C07889=1078.617,151.633,-72.015,174.270,23.846,154.109
C07890=1078.611,151.385,-71.994,174.267,23.844,154.109
C07891=1078.606,151.136,-71.973,174.265,23.841,154.108
C07892=1078.600,150.886,-71.952,174.263,23.840,154.108
C07893=1078.594,150.637,-71.931,174.261,23.837,154.108
C07894=1078.588,150.389,-71.910,174.259,23.835,154.108
C07895=1078.582,150.139,-71.889,174.257,23.832,154.108
C07896=1078.577,149.890,-71.869,174.255,23.830,154.107
C07897=1078.571,149.642,-71.848,174.254,23.828,154.107
C07898=1078.566,149.393,-71.827,174.251,23.825,154.107
C07899=1078.560,149.143,-71.806,174.249,23.823,154.107
C07900=1078.555,148.894,-71.785,174.248,23.821,154.107
C07901=1078.549,148.645,-71.764,174.245,23.818,154.106
C07902=1078.543,148.396,-71.743,174.243,23.816,154.106
C07903=1078.538,148.147,-71.722,174.242,23.814,154.106
C07904=1078.532,147.898,-71.702,174.239,23.811,154.106
C07905=1078.527,147.649,-71.682,174.238,23.810,154.106
C07906=1078.521,147.400,-71.660,174.236,23.807,154.105
C07907=1078.515,147.150,-71.639,174.233,23.805,154.105
C07908=1078.509,146.902,-71.620,174.232,23.802,154.105
C07909=1078.503,146.652,-71.598,174.229,23.800,154.105
C07910=1078.498,146.403,-71.577,174.228,23.798,154.104
C07911=1078.493,146.154,-71.557,174.226,23.795,154.104
C07912=1078.487,145.905,-71.536,174.224,23.793,154.104
C07913=1078.481,145.656,-71.515,174.222,23.791,154.104
C07914=1078.475,145.407,-71.495,174.220,23.788,154.104
C07915=1078.470,145.158,-71.474,174.218,23.786,154.103
C07916=1078.465,144.909,-71.454,174.216,23.784,154.103
C07917=1078.458,144.659,-71.433,174.214,23.781,154.103
C07918=1078.453,144.411,-71.412,174.212,23.779,154.103
C07919=1078.447,144.162,-71.391,174.210,23.777,154.103
C07920=1078.441,143.913,-71.371,174.209,23.774,154.102
C07921=1078.435,143.632,-71.348,174.206,23.772,154.102
C07922=1078.429,143.351,-71.324,174.204,23.769,154.102
C07923=1078.423,143.070,-71.301,174.202,23.767,154.102
C07924=1078.417,142.789,-71.278,174.200,23.764,154.101
C07925=1078.411,142.540,-71.258,174.197,23.761,154.101
C07926=1078.405,142.292,-71.237,174.196,23.759,154.101
C07927=1078.400,142.042,-71.216,174.194,23.757,154.101
C07928=1078.393,141.793,-71.196,174.192,23.755,154.101
C07929=1078.388,141.544,-71.176,174.190,23.752,154.100
C07930=1078.383,141.295,-71.155,174.188,23.750,154.100
C07931=1078.377,141.046,-71.135,174.186,23.748,154.100
C07932=1078.371,140.797,-71.115,174.184,23.745,154.100
C07933=1078.366,140.548,-71.094,174.183,23.743,154.099
C07934=1078.360,140.298,-71.074,174.180,23.741,154.099
C07935=1078.354,140.049,-71.053,174.179,23.738,154.099
C07936=1078.349,139.800,-71.033,174.177,23.736,154.099
C07937=1078.343,139.551,-71.013,174.175,23.734,154.099
C07938=1078.338,139.302,-70.992,174.173,23.731,154.098
C07939=1078.332,139.053,-70.972,174.171,23.729,154.098
C07940=1078.327,138.804,-70.951,174.169,23.726,154.098
C07941=1078.320,138.554,-70.931,174.167,23.724,154.098
C07942=1078.315,138.305,-70.911,174.166,23.722,154.097
C07943=1078.309,138.056,-70.890,174.163,23.720,154.097
C07944=1078.303,137.807,-70.870,174.162,23.717,154.097
C07945=1078.298,137.558,-70.850,174.159,23.715,154.097
C07946=1078.292,137.309,-70.830,174.158,23.713,154.097
C07947=1078.287,137.060,-70.809,174.156,23.711,154.096
C07948=1078.281,136.810,-70.789,174.154,23.708,154.096
C07949=1078.275,136.561,-70.769,174.152,23.706,154.096
C07950=1078.269,136.312,-70.749,174.150,23.703,154.096
C07951=1078.263,136.063,-70.729,174.148,23.701,154.095
C07952=1078.258,135.814,-70.708,174.146,23.699,154.095
C07953=1078.252,135.566,-70.688,174.145,23.696,154.095
C07954=1078.247,135.316,-70.668,174.142,23.694,154.095
C07955=1078.241,135.067,-70.649,174.141,23.692,154.095
C07956=1078.236,134.818,-70.628,174.139,23.689,154.094
C07957=1078.230,134.569,-70.608,174.137,23.687,154.094
C07958=1078.225,134.320,-70.588,174.135,23.685,154.094
C07959=1078.218,134.070,-70.567,174.134,23.682,154.094
C07960=1078.213,133.821,-70.547,174.131,23.680,154.093
C07961=1078.207,133.572,-70.527,174.130,23.678,154.093
C07962=1078.202,133.323,-70.507,174.128,23.675,154.093
C07963=1078.196,133.074,-70.487,174.126,23.673,154.093
C07964=1078.190,132.824,-70.468,174.124,23.671,154.093
C07965=1078.185,132.575,-70.447,174.122,23.668,154.092
C07966=1078.179,132.327,-70.427,174.120,23.666,154.092
C07967=1078.174,132.077,-70.407,174.118,23.663,154.092
C07968=1078.168,131.828,-70.387,174.117,23.661,154.092
C07969=1078.162,131.579,-70.367,174.114,23.659,154.091
C07970=1078.156,131.330,-70.347,174.113,23.657,154.091
C07971=1078.151,131.081,-70.328,174.111,23.654,154.091
C07972=1078.145,130.832,-70.308,174.109,23.652,154.091
C07973=1078.139,130.583,-70.288,174.107,23.649,154.091
C07974=1078.133,130.334,-70.268,174.106,23.648,154.090
C07975=1078.128,130.084,-70.248,174.103,23.645,154.090
C07976=1078.122,129.835,-70.228,174.102,23.642,154.090
C07977=1078.116,129.585,-70.208,174.100,23.640,154.090
C07978=1078.110,129.337,-70.188,174.098,23.638,154.089
C07979=1078.104,129.088,-70.168,174.096,23.636,154.089
C07980=1078.099,128.838,-70.149,174.095,23.633,154.089
C07981=1078.093,128.589,-70.129,174.092,23.631,154.089
C07982=1078.087,128.340,-70.109,174.091,23.629,154.089
C07983=1078.081,128.091,-70.089,174.089,23.626,154.088
C07984=1078.076,127.842,-70.070,174.087,23.624,154.088
C07985=1078.069,127.561,-70.048,174.085,23.621,154.088
C07986=1078.063,127.280,-70.025,174.083,23.619,154.088
C07987=1078.057,126.999,-70.003,174.081,23.616,154.087
C07988=1078.050,126.718,-69.981,174.079,23.613,154.087
C07989=1078.044,126.469,-69.961,174.077,23.611,154.087
C07990=1078.038,126.220,-69.941,174.076,23.609,154.087
C07991=1078.033,125.970,-69.922,174.073,23.607,154.087
C07992=1078.027,125.721,-69.902,174.072,23.604,154.086
C07993=1078.022,125.472,-69.882,174.070,23.602,154.086
C07994=1078.016,125.223,-69.862,174.068,23.600,154.086
C07995=1078.010,124.974,-69.844,174.066,23.597,154.086
C07996=1078.004,124.725,-69.824,174.065,23.595,154.085
C07997=1077.999,124.476,-69.804,174.062,23.592,154.085
C07998=1077.993,124.227,-69.784,174.061,23.590,154.085
C07999=1077.988,123.977,-69.765,174.059,23.588,154.085
C08000=1077.982,123.728,-69.745,174.057,23.585,154.084
C08001=1077.976,123.479,-69.725,174.055,23.583,154.084
C08002=1077.970,123.230,-69.706,174.054,23.581,154.084
C08003=1077.964,122.981,-69.686,174.052,23.578,154.084
C08004=1077.959,122.732,-69.667,174.050,23.576,154.084
C08005=1077.953,122.482,-69.648,174.048,23.573,154.083
C08006=1077.947,122.233,-69.628,174.047,23.571,154.083
C08007=1077.942,121.985,-69.609,174.044,23.569,154.083
C08008=1077.937,121.735,-69.589,174.043,23.566,154.083
C08009=1077.931,121.486,-69.569,174.041,23.564,154.082
C08010=1077.925,121.237,-69.550,174.039,23.561,154.082
C08011=1077.920,120.987,-69.531,174.038,23.559,154.082
C08012=1077.914,120.738,-69.511,174.036,23.557,154.082
C08013=1077.908,120.489,-69.491,174.034,23.554,154.081
C08014=1077.902,120.239,-69.472,174.032,23.552,154.081
C08015=1077.897,119.991,-69.453,174.031,23.550,154.081
C08016=1077.891,119.742,-69.433,174.028,23.547,154.081
C08017=1077.886,119.492,-69.414,174.027,23.545,154.080
C08018=1077.880,119.243,-69.395,174.025,23.542,154.080
C08019=1077.874,118.994,-69.375,174.023,23.540,154.080
C08020=1077.868,118.745,-69.356,174.021,23.537,154.080
C08021=1077.864,118.496,-69.336,174.020,23.535,154.079
C08022=1077.858,118.246,-69.317,174.019,23.533,154.079
C08023=1077.852,117.997,-69.298,174.016,23.530,154.079
C08024=1077.847,117.747,-69.278,174.015,23.528,154.079
C08025=1077.841,117.499,-69.258,174.013,23.526,154.078
C08026=1077.836,117.250,-69.240,174.011,23.523,154.078
C08027=1077.830,117.000,-69.220,174.009,23.520,154.078
C08028=1077.824,116.751,-69.201,174.008,23.518,154.078
C08029=1077.819,116.502,-69.182,174.005,23.516,154.077
C08030=1077.814,116.253,-69.163,174.004,23.513,154.077
C08031=1077.808,116.004,-69.143,174.003,23.511,154.077
C08032=1077.802,115.755,-69.124,174.001,23.508,154.077
C08033=1077.796,115.505,-69.104,173.999,23.506,154.076
C08034=1077.791,115.256,-69.086,173.997,23.504,154.076
C08035=1077.785,115.007,-69.066,173.996,23.501,154.076
C08036=1077.780,114.758,-69.047,173.993,23.499,154.076
C08037=1077.774,114.508,-69.028,173.992,23.496,154.075
C08038=1077.769,114.259,-69.009,173.990,23.493,154.075
C08039=1077.763,114.010,-68.990,173.988,23.492,154.075
C08040=1077.758,113.761,-68.970,173.987,23.489,154.075
C08041=1077.751,113.511,-68.952,173.985,23.486,154.074
C08042=1077.745,113.262,-68.933,173.984,23.485,154.074
C08043=1077.740,113.013,-68.914,173.981,23.482,154.074
C08044=1077.735,112.764,-68.894,173.980,23.479,154.074
C08045=1077.729,112.514,-68.875,173.978,23.477,154.073
C08046=1077.723,112.265,-68.857,173.976,23.475,154.073
C08047=1077.717,112.017,-68.838,173.975,23.472,154.073
C08048=1077.712,111.767,-68.818,173.973,23.470,154.073
C08049=1077.705,111.486,-68.797,173.971,23.467,154.072
C08050=1077.698,111.205,-68.776,173.969,23.464,154.072
C08051=1077.692,110.924,-68.754,173.967,23.462,154.072
C08052=1077.686,110.643,-68.733,173.965,23.459,154.072
C08053=1077.680,110.394,-68.714,173.964,23.457,154.071
C08054=1077.675,110.145,-68.695,173.961,23.454,154.071
C08055=1077.669,109.896,-68.676,173.960,23.452,154.071
C08056=1077.662,109.647,-68.657,173.959,23.450,154.071
C08057=1077.657,109.397,-68.638,173.956,23.447,154.070
C08058=1077.652,109.148,-68.619,173.955,23.445,154.070
C08059=1077.645,108.899,-68.600,173.953,23.442,154.070
C08060=1077.640,108.649,-68.582,173.952,23.440,154.070
C08061=1077.634,108.400,-68.563,173.950,23.438,154.069
C08062=1077.628,108.151,-68.544,173.948,23.435,154.069
C08063=1077.623,107.902,-68.525,173.947,23.433,154.069
C08064=1077.617,107.653,-68.506,173.944,23.430,154.069
C08065=1077.611,107.404,-68.488,173.943,23.428,154.068
C08066=1077.606,107.154,-68.469,173.942,23.426,154.068
C08067=1077.600,106.905,-68.450,173.939,23.423,154.068
C08068=1077.594,106.656,-68.431,173.938,23.421,154.068
C08069=1077.589,106.407,-68.412,173.936,23.418,154.067
C08070=1077.583,106.157,-68.393,173.934,23.416,154.067
C08071=1077.577,105.908,-68.375,173.933,23.414,154.067
C08072=1077.572,105.659,-68.356,173.931,23.411,154.067
C08073=1077.566,105.409,-68.337,173.930,23.408,154.066
C08074=1077.560,105.160,-68.318,173.927,23.406,154.066
C08075=1077.555,104.911,-68.300,173.926,23.404,154.066
C08076=1077.548,104.662,-68.282,173.925,23.401,154.066
C08077=1077.543,104.413,-68.263,173.923,23.399,154.065
C08078=1077.538,104.163,-68.244,173.921,23.396,154.065
C08079=1077.531,103.914,-68.225,173.919,23.394,154.065
C08080=1077.526,103.665,-68.207,173.918,23.392,154.065
C08081=1077.520,103.416,-68.188,173.916,23.389,154.064
C08082=1077.515,103.166,-68.169,173.914,23.386,154.064
C08083=1077.509,102.917,-68.151,173.913,23.384,154.064
C08084=1077.503,102.668,-68.132,173.911,23.382,154.064
C08085=1077.498,102.419,-68.114,173.909,23.379,154.063
C08086=1077.492,102.170,-68.095,173.908,23.377,154.063
C08087=1077.486,101.920,-68.077,173.906,23.374,154.063
C08088=1077.481,101.671,-68.058,173.904,23.372,154.062
C08089=1077.475,101.422,-68.039,173.903,23.369,154.062
C08090=1077.470,101.172,-68.021,173.901,23.367,154.062
C08091=1077.464,100.923,-68.002,173.899,23.365,154.062
C08092=1077.458,100.674,-67.984,173.897,23.362,154.062
C08093=1077.453,100.425,-67.965,173.896,23.360,154.061
C08094=1077.446,100.176,-67.947,173.895,23.357,154.061
C08095=1077.441,99.926,-67.928,173.892,23.355,154.061
C08096=1077.435,99.677,-67.910,173.891,23.353,154.060
C08097=1077.429,99.428,-67.892,173.890,23.350,154.060
C08098=1077.424,99.179,-67.873,173.888,23.347,154.060
C08099=1077.418,98.929,-67.855,173.886,23.346,154.060
C08100=1077.412,98.680,-67.836,173.884,23.343,154.060
C08101=1077.406,98.431,-67.818,173.883,23.340,154.059
C08102=1077.400,98.181,-67.800,173.881,23.338,154.059
C08103=1077.395,97.932,-67.782,173.879,23.335,154.059
C08104=1077.389,97.683,-67.763,173.878,23.333,154.059
C08105=1077.383,97.434,-67.745,173.876,23.331,154.058
C08106=1077.378,97.185,-67.726,173.874,23.328,154.058
C08107=1077.371,96.935,-67.708,173.873,23.326,154.058
C08108=1077.366,96.686,-67.689,173.872,23.323,154.057
C08109=1077.360,96.436,-67.671,173.869,23.321,154.057
C08110=1077.355,96.187,-67.654,173.868,23.319,154.057
C08111=1077.349,95.938,-67.635,173.867,23.316,154.057
C08112=1077.343,95.689,-67.617,173.864,23.314,154.056
C08113=1077.336,95.408,-67.596,173.862,23.311,154.056
C08114=1077.330,95.127,-67.576,173.861,23.308,154.056
C08115=1077.324,94.847,-67.555,173.859,23.305,154.055
C08116=1077.317,94.565,-67.534,173.858,23.303,154.055
C08117=1077.312,94.316,-67.517,173.855,23.300,154.055
C08118=1077.306,94.067,-67.498,173.854,23.298,154.055
C08119=1077.301,93.817,-67.480,173.852,23.295,154.054
C08120=1077.295,93.568,-67.462,173.851,23.293,154.054
C08121=1077.289,93.319,-67.443,173.849,23.291,154.054
C08122=1077.283,93.069,-67.426,173.847,23.288,154.054
C08123=1077.278,92.820,-67.407,173.846,23.285,154.053
C08124=1077.272,92.572,-67.389,173.845,23.283,154.053
C08125=1077.266,92.322,-67.371,173.842,23.280,154.053
C08126=1077.261,92.073,-67.353,173.841,23.278,154.052
C08127=1077.255,91.823,-67.335,173.840,23.275,154.052
C08128=1077.249,91.574,-67.317,173.838,23.273,154.052
C08129=1077.244,91.324,-67.298,173.836,23.270,154.052
C08130=1077.238,91.075,-67.281,173.835,23.268,154.051
C08131=1077.232,90.826,-67.263,173.833,23.266,154.051
C08132=1077.226,90.577,-67.244,173.831,23.263,154.051
C08133=1077.220,90.327,-67.227,173.830,23.261,154.051
C08134=1077.215,90.078,-67.209,173.828,23.258,154.050
C08135=1077.209,89.829,-67.191,173.827,23.256,154.050
C08136=1077.204,89.579,-67.173,173.825,23.254,154.050
C08137=1077.197,89.330,-67.154,173.823,23.251,154.050
C08138=1077.192,89.081,-67.137,173.822,23.249,154.049
C08139=1077.186,88.831,-67.119,173.820,23.246,154.049
C08140=1077.180,88.582,-67.101,173.818,23.243,154.049
C08141=1077.174,88.333,-67.083,173.817,23.241,154.049
C08142=1077.169,88.083,-67.066,173.815,23.239,154.048
C08143=1077.163,87.835,-67.047,173.813,23.236,154.048
C08144=1077.157,87.585,-67.029,173.812,23.234,154.048
C08145=1077.151,87.336,-67.012,173.811,23.232,154.048
C08146=1077.145,87.087,-66.994,173.809,23.229,154.047
C08147=1077.140,86.838,-66.976,173.807,23.226,154.047
C08148=1077.133,86.588,-66.958,173.806,23.224,154.047
C08149=1077.128,86.339,-66.941,173.804,23.221,154.046
C08150=1077.123,86.089,-66.923,173.802,23.219,154.046
C08151=1077.117,85.840,-66.905,173.801,23.217,154.046
C08152=1077.111,85.591,-66.887,173.799,23.214,154.046
C08153=1077.105,85.341,-66.869,173.798,23.212,154.045
C08154=1077.100,85.092,-66.851,173.796,23.209,154.045
C08155=1077.094,84.843,-66.833,173.794,23.206,154.045
C08156=1077.088,84.594,-66.816,173.793,23.204,154.045
C08157=1077.082,84.345,-66.798,173.792,23.202,154.044
C08158=1077.076,84.095,-66.780,173.789,23.199,154.044
C08159=1077.071,83.846,-66.762,173.788,23.196,154.044
C08160=1077.065,83.597,-66.745,173.787,23.195,154.044
C08161=1077.059,83.347,-66.727,173.785,23.192,154.043
C08162=1077.054,83.098,-66.709,173.783,23.189,154.043
C08163=1077.048,82.849,-66.692,173.782,23.187,154.043
C08164=1077.042,82.599,-66.674,173.781,23.185,154.042
C08165=1077.036,82.350,-66.656,173.779,23.182,154.042
C08166=1077.031,82.101,-66.639,173.777,23.179,154.042
C08167=1077.025,81.851,-66.622,173.776,23.177,154.042
C08168=1077.020,81.602,-66.604,173.774,23.174,154.041
C08169=1077.014,81.353,-66.586,173.772,23.172,154.041
C08170=1077.008,81.103,-66.568,173.771,23.169,154.041
C08171=1077.002,80.854,-66.551,173.769,23.167,154.040
C08172=1076.997,80.605,-66.533,173.768,23.164,154.040
C08173=1076.991,80.355,-66.515,173.766,23.162,154.040
C08174=1076.985,80.106,-66.498,173.764,23.159,154.040
C08175=1076.980,79.857,-66.480,173.763,23.157,154.039
C08176=1076.974,79.607,-66.463,173.762,23.154,154.039
C08177=1076.967,79.326,-66.444,173.760,23.151,154.039
C08178=1076.961,79.045,-66.424,173.758,23.149,154.038
C08179=1076.954,78.764,-66.404,173.756,23.146,154.038
C08180=1076.948,78.484,-66.384,173.755,23.143,154.038
C08181=1076.942,78.235,-66.367,173.753,23.140,154.038
C08182=1076.937,77.985,-66.350,173.752,23.138,154.037
C08183=1076.931,77.736,-66.332,173.750,23.136,154.037
C08184=1076.925,77.486,-66.314,173.748,23.133,154.037
C08185=1076.919,77.238,-66.297,173.747,23.130,154.036
C08186=1076.913,76.989,-66.280,173.746,23.128,154.036
C08187=1076.908,76.738,-66.262,173.743,23.125,154.036
C08188=1076.902,76.489,-66.245,173.742,23.123,154.036
C08189=1076.897,76.240,-66.227,173.741,23.121,154.035
C08190=1076.890,75.991,-66.210,173.739,23.119,154.035
C08191=1076.884,75.741,-66.193,173.737,23.116,154.035
C08192=1076.879,75.492,-66.176,173.736,23.113,154.035
C08193=1076.873,75.243,-66.158,173.735,23.111,154.034
C08194=1076.867,74.993,-66.141,173.733,23.108,154.034
C08195=1076.861,74.744,-66.124,173.731,23.106,154.034
C08196=1076.856,74.495,-66.106,173.730,23.103,154.033
C08197=1076.850,74.246,-66.089,173.729,23.101,154.033
C08198=1076.844,73.996,-66.072,173.727,23.098,154.033
C08199=1076.838,73.747,-66.054,173.725,23.096,154.033
C08200=1076.833,73.498,-66.037,173.724,23.093,154.032
C08201=1076.828,73.248,-66.020,173.722,23.091,154.032
C08202=1076.821,72.999,-66.003,173.721,23.088,154.032
C08203=1076.815,72.749,-65.986,173.719,23.086,154.031
C08204=1076.810,72.500,-65.968,173.718,23.083,154.031
C08205=1076.804,72.251,-65.951,173.716,23.081,154.031
C08206=1076.798,72.001,-65.934,173.715,23.078,154.031
C08207=1076.792,71.752,-65.917,173.713,23.076,154.030
C08208=1076.787,71.502,-65.900,173.711,23.073,154.030
C08209=1076.781,71.253,-65.883,173.710,23.070,154.030
C08210=1076.775,71.004,-65.865,173.709,23.068,154.029
C08211=1076.770,70.754,-65.848,173.707,23.066,154.029
C08212=1076.763,70.505,-65.831,173.705,23.063,154.029
C08213=1076.758,70.256,-65.814,173.704,23.060,154.029
C08214=1076.753,70.006,-65.797,173.703,23.058,154.028
C08215=1076.747,69.757,-65.780,173.700,23.056,154.028
C08216=1076.741,69.508,-65.763,173.699,23.053,154.028
C08217=1076.735,69.258,-65.746,173.698,23.051,154.028
C08218=1076.729,69.009,-65.729,173.696,23.049,154.027
C08219=1076.724,68.759,-65.712,173.694,23.046,154.027
C08220=1076.718,68.511,-65.695,173.693,23.043,154.027
C08221=1076.712,68.261,-65.678,173.692,23.041,154.026
C08222=1076.705,68.012,-65.661,173.691,23.039,154.026
C08223=1076.700,67.762,-65.644,173.688,23.036,154.026
C08224=1076.694,67.513,-65.627,173.687,23.033,154.026
C08225=1076.689,67.263,-65.610,173.686,23.031,154.025
C08226=1076.683,67.015,-65.593,173.684,23.028,154.025
C08227=1076.677,66.765,-65.576,173.682,23.026,154.025
C08228=1076.670,66.516,-65.559,173.681,23.023,154.025
C08229=1076.665,66.266,-65.542,173.680,23.021,154.024
C08230=1076.660,66.016,-65.525,173.678,23.018,154.024
C08231=1076.654,65.768,-65.508,173.676,23.016,154.024
C08232=1076.649,65.518,-65.491,173.675,23.013,154.023
C08233=1076.642,65.269,-65.474,173.674,23.011,154.023
C08234=1076.637,65.020,-65.457,173.672,23.008,154.023
C08235=1076.631,64.770,-65.441,173.670,23.006,154.023
C08236=1076.625,64.520,-65.423,173.669,23.003,154.022
C08237=1076.619,64.271,-65.407,173.668,23.001,154.022
C08238=1076.613,64.022,-65.391,173.666,22.998,154.022
C08239=1076.608,63.773,-65.373,173.665,22.996,154.021
C08240=1076.602,63.523,-65.357,173.663,22.993,154.021
C08241=1076.595,63.242,-65.338,173.661,22.990,154.021
C08242=1076.588,62.961,-65.319,173.660,22.988,154.021
C08243=1076.581,62.680,-65.300,173.658,22.985,154.020
C08244=1076.575,62.399,-65.281,173.657,22.982,154.020
C08245=1076.569,62.150,-65.265,173.654,22.979,154.020
C08246=1076.563,61.901,-65.249,173.653,22.977,154.019
C08247=1076.557,61.651,-65.231,173.652,22.975,154.019
C08248=1076.551,61.402,-65.215,173.650,22.973,154.019
C08249=1076.545,61.152,-65.198,173.648,22.970,154.019
C08250=1076.540,60.902,-65.181,173.647,22.967,154.018
C08251=1076.533,60.654,-65.164,173.646,22.965,154.018
C08252=1076.527,60.404,-65.148,173.645,22.963,154.018
C08253=1076.521,60.155,-65.132,173.642,22.960,154.018
C08254=1076.516,59.905,-65.115,173.641,22.957,154.017
C08255=1076.510,59.656,-65.099,173.640,22.955,154.017
C08256=1076.504,59.407,-65.082,173.639,22.952,154.017
C08257=1076.498,59.158,-65.066,173.636,22.950,154.016
C08258=1076.492,58.908,-65.048,173.635,22.947,154.016
C08259=1076.486,58.658,-65.032,173.634,22.945,154.016
C08260=1076.480,58.409,-65.016,173.633,22.942,154.016
C08261=1076.474,58.160,-64.999,173.630,22.940,154.015
C08262=1076.469,57.910,-64.982,173.629,22.937,154.015
C08263=1076.463,57.661,-64.966,173.628,22.935,154.015
C08264=1076.457,57.412,-64.949,173.627,22.933,154.015
C08265=1076.451,57.162,-64.933,173.624,22.930,154.014
C08266=1076.446,56.913,-64.916,173.623,22.928,154.014
C08267=1076.440,56.663,-64.900,173.622,22.925,154.014
C08268=1076.434,56.414,-64.884,173.621,22.923,154.013
C08269=1076.428,56.165,-64.868,173.618,22.920,154.013
C08270=1076.423,55.915,-64.851,173.617,22.918,154.013
C08271=1076.416,55.666,-64.834,173.616,22.915,154.013
C08272=1076.410,55.417,-64.818,173.615,22.913,154.012
C08273=1076.405,55.168,-64.801,173.612,22.910,154.012
C08274=1076.399,54.918,-64.785,173.611,22.907,154.012
C08275=1076.393,54.669,-64.768,173.610,22.905,154.011
C08276=1076.387,54.419,-64.752,173.609,22.903,154.011
C08277=1076.381,54.170,-64.736,173.607,22.900,154.011
C08278=1076.376,53.921,-64.719,173.605,22.897,154.011
C08279=1076.370,53.671,-64.703,173.604,22.895,154.010
C08280=1076.364,53.422,-64.686,173.603,22.893,154.010
C08281=1076.358,53.172,-64.670,173.601,22.890,154.010
C08282=1076.352,52.923,-64.654,173.599,22.887,154.009
C08283=1076.347,52.674,-64.638,173.598,22.885,154.009
C08284=1076.341,52.424,-64.621,173.597,22.882,154.009
C08285=1076.335,52.175,-64.605,173.596,22.880,154.008
C08286=1076.329,51.925,-64.588,173.594,22.877,154.008
C08287=1076.323,51.676,-64.572,173.592,22.874,154.008
C08288=1076.317,51.426,-64.556,173.591,22.872,154.008
C08289=1076.312,51.177,-64.540,173.590,22.869,154.007
C08290=1076.306,50.927,-64.524,173.588,22.867,154.007
C08291=1076.300,50.678,-64.508,173.586,22.864,154.007
C08292=1076.295,50.428,-64.491,173.585,22.862,154.006
C08293=1076.289,50.179,-64.474,173.584,22.859,154.006
C08294=1076.283,49.930,-64.459,173.582,22.857,154.006
C08295=1076.277,49.681,-64.442,173.581,22.854,154.006
C08296=1076.272,49.431,-64.426,173.579,22.852,154.005
C08297=1076.266,49.182,-64.410,173.578,22.849,154.005
C08298=1076.260,48.932,-64.394,173.577,22.847,154.005
C08299=1076.255,48.682,-64.377,173.575,22.844,154.005
C08300=1076.249,48.433,-64.361,173.573,22.842,154.004
C08301=1076.243,48.184,-64.345,173.572,22.839,154.004
C08302=1076.237,47.934,-64.329,173.571,22.837,154.004
C08303=1076.232,47.686,-64.313,173.569,22.834,154.003
C08304=1076.226,47.436,-64.297,173.568,22.831,154.003
C08305=1076.219,47.155,-64.278,173.566,22.829,154.003
C08306=1076.213,46.873,-64.260,173.564,22.825,154.002
C08307=1076.207,46.592,-64.242,173.563,22.823,154.002
C08308=1076.200,46.310,-64.224,173.561,22.820,154.002
C08309=1076.194,46.061,-64.208,173.560,22.817,154.001
C08310=1076.189,45.812,-64.192,173.559,22.815,154.001
C08311=1076.183,45.563,-64.176,173.557,22.812,154.001
C08312=1076.178,45.313,-64.160,173.555,22.809,154.000
C08313=1076.172,45.064,-64.144,173.554,22.807,154.000
C08314=1076.166,44.814,-64.128,173.553,22.804,154.000
C08315=1076.160,44.565,-64.111,173.552,22.802,154.000
C08316=1076.154,44.315,-64.096,173.549,22.799,153.999
C08317=1076.149,44.067,-64.080,173.548,22.797,153.999
C08318=1076.143,43.817,-64.064,173.547,22.794,153.999
C08319=1076.137,43.567,-64.048,173.546,22.791,153.998
C08320=1076.131,43.318,-64.032,173.545,22.789,153.998
C08321=1076.125,43.069,-64.016,173.542,22.786,153.998
C08322=1076.120,42.819,-64.000,173.541,22.784,153.998
C08323=1076.114,42.570,-63.984,173.540,22.781,153.997
C08324=1076.108,42.321,-63.968,173.539,22.779,153.997
C08325=1076.103,42.071,-63.952,173.537,22.776,153.997
C08326=1076.097,41.821,-63.936,173.535,22.774,153.996
C08327=1076.091,41.571,-63.921,173.534,22.771,153.996
C08328=1076.084,41.322,-63.905,173.533,22.769,153.996
C08329=1076.079,41.074,-63.889,173.532,22.766,153.996
C08330=1076.073,40.824,-63.874,173.529,22.763,153.995
C08331=1076.067,40.574,-63.857,173.528,22.761,153.995
C08332=1076.062,40.324,-63.842,173.527,22.759,153.995
C08333=1076.056,40.075,-63.825,173.526,22.756,153.994
C08334=1076.050,39.826,-63.810,173.524,22.754,153.994
C08335=1076.045,39.576,-63.794,173.522,22.751,153.994
C08336=1076.038,39.327,-63.778,173.521,22.748,153.994
C08337=1076.032,39.077,-63.763,173.520,22.746,153.993
C08338=1076.026,38.828,-63.747,173.519,22.744,153.993
C08339=1076.021,38.579,-63.731,173.517,22.741,153.993
C08340=1076.016,38.329,-63.715,173.515,22.738,153.992
C08341=1076.010,38.079,-63.700,173.514,22.736,153.992
C08342=1076.003,37.830,-63.684,173.513,22.733,153.992
C08343=1075.998,37.581,-63.669,173.511,22.731,153.992
C08344=1075.992,37.332,-63.653,173.510,22.729,153.991
C08345=1075.987,37.082,-63.637,173.508,22.726,153.991
C08346=1075.980,36.833,-63.621,173.507,22.723,153.991
C08347=1075.974,36.583,-63.606,173.506,22.721,153.990
C08348=1075.969,36.334,-63.590,173.504,22.718,153.990
C08349=1075.962,36.084,-63.575,173.503,22.716,153.990
C08350=1075.957,35.834,-63.559,173.501,22.713,153.990
C08351=1075.951,35.585,-63.543,173.500,22.711,153.989
C08352=1075.945,35.336,-63.529,173.498,22.708,153.989
C08353=1075.939,35.087,-63.512,173.497,22.706,153.989
C08354=1075.933,34.837,-63.497,173.496,22.704,153.988
C08355=1075.927,34.588,-63.481,173.494,22.701,153.988
C08356=1075.921,34.338,-63.466,173.493,22.698,153.988
C08357=1075.916,34.089,-63.450,173.491,22.696,153.988
C08358=1075.909,33.840,-63.435,173.490,22.693,153.987
C08359=1075.904,33.590,-63.419,173.489,22.691,153.987
C08360=1075.899,33.340,-63.404,173.487,22.688,153.987
C08361=1075.892,33.091,-63.388,173.485,22.686,153.986
C08362=1075.886,32.841,-63.373,173.484,22.683,153.986
C08363=1075.881,32.591,-63.357,173.483,22.681,153.986
C08364=1075.875,32.343,-63.342,173.482,22.678,153.986
C08365=1075.869,32.093,-63.326,173.480,22.676,153.985
C08366=1075.863,31.843,-63.312,173.478,22.673,153.985
C08367=1075.857,31.595,-63.296,173.477,22.671,153.985
C08368=1075.852,31.345,-63.280,173.476,22.668,153.984
C08369=1075.845,31.063,-63.263,173.474,22.665,153.984
C08370=1075.838,30.782,-63.246,173.473,22.662,153.984
C08371=1075.832,30.502,-63.229,173.471,22.660,153.984
C08372=1075.825,30.220,-63.211,173.470,22.657,153.983
C08373=1075.819,29.970,-63.196,173.468,22.654,153.983
C08374=1075.814,29.721,-63.180,173.467,22.652,153.983
C08375=1075.808,29.472,-63.164,173.465,22.649,153.982
C08376=1075.802,29.223,-63.150,173.464,22.646,153.982
C08377=1075.796,28.973,-63.134,173.462,22.644,153.982
C08378=1075.790,28.723,-63.119,173.461,22.642,153.981
C08379=1075.785,28.474,-63.104,173.460,22.639,153.981
C08380=1075.778,28.225,-63.088,173.458,22.636,153.981
C08381=1075.773,27.975,-63.073,173.457,22.634,153.981
C08382=1075.766,27.725,-63.058,173.455,22.631,153.980
C08383=1075.761,27.476,-63.043,173.454,22.630,153.980
C08384=1075.755,27.226,-63.028,173.453,22.627,153.980
C08385=1075.750,26.977,-63.012,173.451,22.624,153.980
C08386=1075.743,26.728,-62.997,173.449,22.622,153.979
C08387=1075.737,26.478,-62.981,173.448,22.619,153.979
C08388=1075.732,26.229,-62.967,173.447,22.617,153.979
C08389=1075.725,25.979,-62.952,173.446,22.615,153.978
C08390=1075.720,25.729,-62.936,173.444,22.612,153.978
C08391=1075.714,25.480,-62.922,173.442,22.609,153.978
C08392=1075.708,25.230,-62.906,173.441,22.607,153.978
C08393=1075.702,24.981,-62.891,173.440,22.604,153.977
C08394=1075.696,24.732,-62.875,173.439,22.602,153.977
C08395=1075.690,24.482,-62.860,173.437,22.599,153.977
C08396=1075.684,24.233,-62.845,173.435,22.597,153.976
C08397=1075.679,23.983,-62.830,173.434,22.594,153.976
C08398=1075.672,23.734,-62.815,173.433,22.592,153.976
C08399=1075.667,23.485,-62.800,173.431,22.589,153.976
C08400=1075.661,23.235,-62.785,173.430,22.587,153.975
C08401=1075.654,22.985,-62.770,173.429,22.584,153.975
C08402=1075.649,22.736,-62.755,173.427,22.582,153.975
C08403=1075.643,22.486,-62.740,173.426,22.579,153.974
C08404=1075.638,22.237,-62.725,173.424,22.577,153.974
C08405=1075.632,21.987,-62.710,173.423,22.574,153.974
C08406=1075.625,21.738,-62.695,173.422,22.572,153.974
C08407=1075.620,21.488,-62.680,173.420,22.569,153.973
C08408=1075.614,21.239,-62.665,173.419,22.567,153.973
C08409=1075.608,20.990,-62.650,173.417,22.564,153.973
C08410=1075.602,20.740,-62.635,173.416,22.562,153.972
C08411=1075.597,20.491,-62.620,173.415,22.559,153.972
C08412=1075.590,20.241,-62.605,173.414,22.557,153.972
C08413=1075.585,19.992,-62.590,173.411,22.554,153.972
C08414=1075.579,19.742,-62.575,173.410,22.552,153.972
C08415=1075.573,19.492,-62.561,173.409,22.550,153.971
C08416=1075.568,19.243,-62.546,173.408,22.547,153.971
C08417=1075.561,18.993,-62.531,173.406,22.545,153.971
C08418=1075.556,18.744,-62.516,173.405,22.542,153.970
C08419=1075.549,18.495,-62.501,173.403,22.539,153.970
C08420=1075.544,18.245,-62.486,173.402,22.537,153.970
C08421=1075.538,17.996,-62.471,173.401,22.535,153.970
C08422=1075.532,17.747,-62.457,173.399,22.532,153.969
C08423=1075.526,17.497,-62.442,173.398,22.530,153.969
C08424=1075.520,17.246,-62.427,173.397,22.527,153.969
C08425=1075.514,16.997,-62.412,173.395,22.524,153.968
C08426=1075.508,16.748,-62.397,173.394,22.522,153.968
C08427=1075.502,16.499,-62.383,173.392,22.519,153.968
C08428=1075.496,16.249,-62.368,173.391,22.518,153.968
C08429=1075.491,16.000,-62.353,173.390,22.515,153.967
C08430=1075.485,15.750,-62.338,173.388,22.513,153.967
C08431=1075.479,15.501,-62.324,173.386,22.510,153.967
C08432=1075.473,15.251,-62.309,173.385,22.507,153.967
C08433=1075.467,14.971,-62.292,173.384,22.504,153.966
C08434=1075.460,14.691,-62.276,173.382,22.502,153.966
C08435=1075.453,14.412,-62.259,173.381,22.499,153.966
C08436=1075.446,14.132,-62.243,173.379,22.496,153.965
C08437=1075.441,13.882,-62.228,173.377,22.494,153.965
C08438=1075.435,13.633,-62.214,173.376,22.491,153.965
C08439=1075.429,13.383,-62.199,173.375,22.489,153.964
C08440=1075.423,13.134,-62.184,173.374,22.486,153.964
C08441=1075.417,12.884,-62.169,173.372,22.484,153.964
C08442=1075.411,12.635,-62.155,173.370,22.482,153.964
C08443=1075.405,12.385,-62.140,173.369,22.479,153.963
C08444=1075.399,12.136,-62.126,173.368,22.477,153.963
C08445=1075.393,11.886,-62.112,173.366,22.474,153.963
C08446=1075.387,11.637,-62.097,173.365,22.472,153.963
C08447=1075.381,11.387,-62.082,173.364,22.469,153.962
C08448=1075.375,11.138,-62.068,173.362,22.467,153.962
C08449=1075.369,10.888,-62.053,173.360,22.465,153.962
C08450=1075.363,10.639,-62.039,173.359,22.462,153.962
C08451=1075.357,10.389,-62.024,173.358,22.460,153.961
C08452=1075.351,10.140,-62.010,173.357,22.457,153.961
C08453=1075.345,9.890,-61.995,173.356,22.455,153.961
C08454=1075.340,9.641,-61.981,173.353,22.452,153.961
C08455=1075.333,9.391,-61.966,173.352,22.450,153.960
C08456=1075.328,9.142,-61.952,173.351,22.448,153.960
C08457=1075.321,8.892,-61.937,173.350,22.445,153.960
C08458=1075.316,8.643,-61.923,173.348,22.443,153.959
C08459=1075.310,8.393,-61.909,173.347,22.440,153.959
C08460=1075.304,8.144,-61.894,173.346,22.438,153.959
C08461=1075.298,7.894,-61.880,173.344,22.435,153.959
C08462=1075.292,7.644,-61.865,173.342,22.433,153.958
C08463=1075.286,7.395,-61.851,173.341,22.431,153.958
C08464=1075.280,7.146,-61.837,173.340,22.428,153.958
C08465=1075.274,6.896,-61.823,173.339,22.426,153.958
C08466=1075.268,6.647,-61.808,173.337,22.423,153.957
C08467=1075.262,6.397,-61.794,173.335,22.420,153.957
C08468=1075.256,6.148,-61.780,173.334,22.418,153.957
C08469=1075.251,5.898,-61.766,173.333,22.416,153.957
C08470=1075.244,5.649,-61.751,173.332,22.414,153.956
C08471=1075.239,5.399,-61.737,173.330,22.411,153.956
C08472=1075.232,5.149,-61.722,173.329,22.409,153.956
C08473=1075.227,4.900,-61.708,173.327,22.406,153.956
C08474=1075.221,4.651,-61.694,173.326,22.403,153.955
C08475=1075.215,4.400,-61.679,173.325,22.401,153.955
C08476=1075.209,4.152,-61.665,173.323,22.399,153.955
C08477=1075.204,3.902,-61.651,173.322,22.397,153.954
C08478=1075.197,3.652,-61.636,173.321,22.394,153.954
C08479=1075.192,3.403,-61.622,173.319,22.392,153.954
C08480=1075.186,3.153,-61.609,173.317,22.389,153.954
C08481=1075.179,2.904,-61.594,173.316,22.386,153.953
C08482=1075.174,2.654,-61.580,173.315,22.384,153.953
C08483=1075.168,2.405,-61.565,173.313,22.382,153.953
C08484=1075.162,2.155,-61.551,173.312,22.380,153.953
C08485=1075.157,1.905,-61.537,173.311,22.377,153.952
C08486=1075.151,1.656,-61.523,173.309,22.374,153.952
C08487=1075.145,1.406,-61.509,173.308,22.372,153.952
C08488=1075.139,1.157,-61.495,173.306,22.369,153.952
C08489=1075.133,0.908,-61.480,173.305,22.367,153.951
C08490=1075.127,0.658,-61.466,173.304,22.365,153.951
C08491=1075.121,0.409,-61.452,173.303,22.363,153.951
C08492=1075.115,0.159,-61.438,173.301,22.360,153.950
C08493=1075.110,-0.090,-61.424,173.299,22.357,153.950
C08494=1075.104,-0.341,-61.410,173.298,22.355,153.950
C08495=1075.098,-0.590,-61.395,173.297,22.352,153.950
C08496=1075.093,-0.839,-61.381,173.296,22.350,153.949
C08497=1075.085,-1.117,-61.366,173.294,22.347,153.949
C08498=1075.079,-1.395,-61.350,173.292,22.345,153.949
C08499=1075.073,-1.672,-61.334,173.291,22.342,153.949
C08500=1075.066,-1.951,-61.319,173.289,22.339,153.948
C08501=1075.061,-2.200,-61.304,173.288,22.337,153.948
C08502=1075.054,-2.449,-61.291,173.287,22.334,153.948
C08503=1075.049,-2.699,-61.277,173.285,22.332,153.947
C08504=1075.043,-2.949,-61.263,173.284,22.329,153.947
C08505=1075.037,-3.198,-61.248,173.283,22.327,153.947
C08506=1075.032,-3.448,-61.235,173.281,22.325,153.947
C08507=1075.025,-3.697,-61.221,173.279,22.322,153.946
C08508=1075.019,-3.947,-61.207,173.278,22.320,153.946
C08509=1075.014,-4.197,-61.193,173.277,22.318,153.946
C08510=1075.007,-4.446,-61.179,173.276,22.315,153.946
C08511=1075.001,-4.696,-61.165,173.274,22.313,153.945
C08512=1074.995,-4.945,-61.152,173.273,22.310,153.945
C08513=1074.990,-5.195,-61.138,173.271,22.308,153.945
C08514=1074.984,-5.444,-61.124,173.270,22.306,153.945
C08515=1074.977,-5.694,-61.110,173.268,22.303,153.944
C08516=1074.972,-5.943,-61.096,173.267,22.301,153.944
C08517=1074.965,-6.192,-61.083,173.266,22.299,153.944
C08518=1074.959,-6.443,-61.068,173.265,22.296,153.944
C08519=1074.954,-6.692,-61.054,173.263,22.294,153.943
C08520=1074.948,-6.942,-61.041,173.261,22.292,153.943
C08521=1074.942,-7.191,-61.027,173.260,22.289,153.943
C08522=1074.935,-7.441,-61.014,173.259,22.287,153.943
C08523=1074.930,-7.691,-61.000,173.257,22.285,153.943
C08524=1074.924,-7.940,-60.986,173.256,22.282,153.942
C08525=1074.918,-8.189,-60.972,173.255,22.280,153.942
C08526=1074.912,-8.438,-60.958,173.254,22.277,153.942
C08527=1074.905,-8.688,-60.944,173.251,22.275,153.942
C08528=1074.900,-8.938,-60.931,173.250,22.273,153.941
C08529=1074.894,-9.187,-60.917,173.249,22.270,153.941
C08530=1074.888,-9.437,-60.903,173.248,22.268,153.941
C08531=1074.883,-9.686,-60.890,173.246,22.266,153.941
C08532=1074.876,-9.936,-60.876,173.245,22.263,153.940
C08533=1074.871,-10.186,-60.862,173.244,22.261,153.940
C08534=1074.864,-10.435,-60.849,173.242,22.259,153.940
C08535=1074.859,-10.685,-60.835,173.240,22.256,153.940
C08536=1074.853,-10.934,-60.822,173.239,22.254,153.939
C08537=1074.847,-11.184,-60.808,173.238,22.252,153.939
C08538=1074.840,-11.434,-60.794,173.237,22.249,153.939
C08539=1074.835,-11.683,-60.780,173.235,22.247,153.939
C08540=1074.829,-11.932,-60.767,173.234,22.245,153.938
C08541=1074.823,-12.182,-60.753,173.232,22.242,153.938
C08542=1074.817,-12.431,-60.740,173.231,22.240,153.938
C08543=1074.812,-12.681,-60.727,173.229,22.238,153.938
C08544=1074.805,-12.931,-60.713,173.228,22.235,153.937
C08545=1074.799,-13.181,-60.699,173.227,22.233,153.937
C08546=1074.794,-13.431,-60.685,173.226,22.230,153.937
C08547=1074.788,-13.680,-60.672,173.224,22.228,153.937
C08548=1074.782,-13.929,-60.658,173.222,22.225,153.936
C08549=1074.776,-14.179,-60.645,173.221,22.223,153.936
C08550=1074.771,-14.428,-60.631,173.220,22.221,153.936
C08551=1074.764,-14.678,-60.618,173.218,22.219,153.936
C08552=1074.759,-14.927,-60.604,173.217,22.216,153.935
C08553=1074.752,-15.178,-60.591,173.216,22.214,153.935
C08554=1074.746,-15.427,-60.578,173.214,22.212,153.935
C08555=1074.741,-15.677,-60.564,173.213,22.210,153.935
C08556=1074.735,-15.926,-60.551,173.211,22.207,153.935
C08557=1074.728,-16.175,-60.537,173.210,22.205,153.934
C08558=1074.723,-16.425,-60.524,173.208,22.203,153.934
C08559=1074.717,-16.675,-60.511,173.207,22.200,153.934
C08560=1074.710,-16.924,-60.497,173.206,22.198,153.934
C08561=1074.703,-17.200,-60.482,173.204,22.195,153.933
C08562=1074.697,-17.477,-60.468,173.202,22.193,153.933
C08563=1074.691,-17.753,-60.453,173.201,22.190,153.933
C08564=1074.685,-18.029,-60.438,173.199,22.188,153.933
C08565=1074.678,-18.279,-60.425,173.198,22.186,153.932
C08566=1074.672,-18.528,-60.411,173.197,22.183,153.932
C08567=1074.665,-18.777,-60.398,173.195,22.181,153.932
C08568=1074.660,-19.028,-60.385,173.194,22.179,153.932
C08569=1074.654,-19.277,-60.372,173.193,22.176,153.931
C08570=1074.648,-19.526,-60.358,173.191,22.174,153.931
C08571=1074.642,-19.776,-60.345,173.189,22.172,153.931
C08572=1074.636,-20.026,-60.332,173.188,22.170,153.931
C08573=1074.630,-20.275,-60.319,173.187,22.167,153.931
C08574=1074.624,-20.524,-60.306,173.185,22.165,153.930
C08575=1074.619,-20.774,-60.292,173.184,22.163,153.930
C08576=1074.613,-21.024,-60.279,173.183,22.160,153.930
C08577=1074.606,-21.273,-60.266,173.181,22.158,153.930
C08578=1074.601,-21.524,-60.252,173.180,22.156,153.929
C08579=1074.594,-21.773,-60.239,173.178,22.154,153.929
C08580=1074.588,-22.022,-60.226,173.177,22.151,153.929
C08581=1074.582,-22.272,-60.213,173.175,22.149,153.929
C08582=1074.577,-22.522,-60.199,173.174,22.147,153.929
C08583=1074.571,-22.771,-60.186,173.173,22.145,153.928
C08584=1074.565,-23.021,-60.174,173.172,22.142,153.928
C08585=1074.558,-23.270,-60.160,173.170,22.140,153.928
C08586=1074.553,-23.520,-60.146,173.169,22.138,153.928
C08587=1074.547,-23.770,-60.134,173.167,22.135,153.927
C08588=1074.541,-24.019,-60.121,173.166,22.133,153.927
C08589=1074.535,-24.269,-60.108,173.164,22.131,153.927
C08590=1074.530,-24.518,-60.094,173.163,22.129,153.927
C08591=1074.524,-24.768,-60.082,173.162,22.126,153.927
C08592=1074.517,-25.018,-60.068,173.160,22.124,153.926
C08593=1074.511,-25.267,-60.055,173.159,22.122,153.926
C08594=1074.505,-25.517,-60.043,173.158,22.120,153.926
C08595=1074.500,-25.766,-60.029,173.156,22.117,153.926
C08596=1074.494,-26.016,-60.016,173.154,22.115,153.926
C08597=1074.488,-26.265,-60.003,173.153,22.113,153.925
C08598=1074.482,-26.515,-59.991,173.152,22.111,153.925
C08599=1074.476,-26.764,-59.977,173.150,22.108,153.925
C08600=1074.471,-27.014,-59.964,173.149,22.106,153.925
C08601=1074.465,-27.263,-59.951,173.148,22.104,153.924
C08602=1074.459,-27.513,-59.938,173.146,22.102,153.924
C08603=1074.453,-27.762,-59.925,173.144,22.099,153.924
C08604=1074.447,-28.012,-59.913,173.143,22.097,153.924
C08605=1074.441,-28.262,-59.899,173.142,22.095,153.924
C08606=1074.435,-28.511,-59.887,173.140,22.093,153.923
C08607=1074.428,-28.761,-59.873,173.139,22.091,153.923
C08608=1074.422,-29.011,-59.861,173.138,22.088,153.923
C08609=1074.417,-29.260,-59.848,173.136,22.086,153.923
C08610=1074.410,-29.510,-59.835,173.135,22.085,153.923
C08611=1074.404,-29.760,-59.823,173.133,22.082,153.922
C08612=1074.398,-30.009,-59.809,173.132,22.080,153.922
C08613=1074.392,-30.259,-59.797,173.130,22.077,153.922
C08614=1074.386,-30.508,-59.783,173.129,22.075,153.922
C08615=1074.380,-30.758,-59.771,173.128,22.073,153.922
C08616=1074.374,-31.008,-59.758,173.126,22.071,153.921
C08617=1074.368,-31.257,-59.745,173.125,22.069,153.921
C08618=1074.362,-31.507,-59.733,173.124,22.067,153.921
C08619=1074.356,-31.757,-59.720,173.122,22.065,153.921
C08620=1074.350,-32.006,-59.707,173.120,22.062,153.921
C08621=1074.344,-32.256,-59.694,173.119,22.060,153.920
C08622=1074.338,-32.506,-59.682,173.118,22.058,153.920
C08623=1074.333,-32.754,-59.669,173.116,22.055,153.920
C08624=1074.327,-33.004,-59.656,173.115,22.054,153.920
C08625=1074.319,-33.280,-59.642,173.114,22.052,153.920
C08626=1074.313,-33.555,-59.627,173.111,22.049,153.919
C08627=1074.306,-33.831,-59.614,173.110,22.046,153.919
C08628=1074.299,-34.106,-59.600,173.109,22.044,153.919
C08629=1074.294,-34.356,-59.588,173.108,22.042,153.919
C08630=1074.287,-34.605,-59.574,173.105,22.039,153.919
C08631=1074.282,-34.854,-59.562,173.104,22.038,153.918
C08632=1074.276,-35.104,-59.550,173.103,22.035,153.918
C08633=1074.270,-35.354,-59.536,173.101,22.033,153.918
C08634=1074.264,-35.603,-59.524,173.100,22.031,153.918
C08635=1074.258,-35.853,-59.511,173.099,22.029,153.917
C08636=1074.252,-36.103,-59.499,173.097,22.027,153.917
C08637=1074.246,-36.353,-59.486,173.096,22.025,153.917
C08638=1074.241,-36.602,-59.473,173.094,22.022,153.917
C08639=1074.235,-36.852,-59.461,173.093,22.020,153.917
C08640=1074.229,-37.101,-59.448,173.091,22.018,153.917
C08641=1074.223,-37.351,-59.436,173.090,22.016,153.916
C08642=1074.216,-37.600,-59.423,173.089,22.014,153.916
C08643=1074.210,-37.850,-59.410,173.087,22.011,153.916
C08644=1074.205,-38.099,-59.398,173.086,22.009,153.916
C08645=1074.199,-38.349,-59.386,173.085,22.007,153.916
C08646=1074.193,-38.599,-59.373,173.083,22.006,153.915
C08647=1074.187,-38.849,-59.361,173.082,22.003,153.915
C08648=1074.181,-39.099,-59.348,173.080,22.001,153.915
C08649=1074.174,-39.348,-59.335,173.078,21.999,153.915
C08650=1074.169,-39.597,-59.323,173.077,21.997,153.915
C08651=1074.163,-39.847,-59.311,173.076,21.994,153.914
C08652=1074.157,-40.097,-59.298,173.074,21.992,153.914
C08653=1074.150,-40.346,-59.286,173.073,21.990,153.914
C08654=1074.145,-40.596,-59.274,173.072,21.989,153.914
C08655=1074.139,-40.846,-59.261,173.070,21.987,153.914
C08656=1074.133,-41.095,-59.249,173.069,21.984,153.914
C08657=1074.127,-41.345,-59.237,173.067,21.982,153.913
C08658=1074.120,-41.594,-59.224,173.065,21.980,153.913
C08659=1074.115,-41.844,-59.211,173.064,21.978,153.913
C08660=1074.108,-42.094,-59.199,173.063,21.976,153.913
C08661=1074.103,-42.343,-59.187,173.061,21.974,153.913
C08662=1074.097,-42.593,-59.174,173.060,21.972,153.913
C08663=1074.090,-42.842,-59.162,173.059,21.970,153.912
C08664=1074.084,-43.092,-59.150,173.057,21.968,153.912
C08665=1074.078,-43.342,-59.137,173.056,21.966,153.912
C08666=1074.073,-43.591,-59.125,173.055,21.964,153.912
C08667=1074.066,-43.841,-59.113,173.052,21.961,153.912
C08668=1074.060,-44.091,-59.101,173.051,21.959,153.912
C08669=1074.054,-44.341,-59.088,173.050,21.957,153.911
C08670=1074.048,-44.590,-59.076,173.048,21.955,153.911
C08671=1074.043,-44.839,-59.064,173.047,21.953,153.911
C08672=1074.037,-45.089,-59.051,173.046,21.951,153.911
C08673=1074.030,-45.339,-59.039,173.044,21.949,153.911
C08674=1074.024,-45.589,-59.027,173.043,21.947,153.910
C08675=1074.019,-45.838,-59.015,173.042,21.945,153.910
C08676=1074.012,-46.087,-59.003,173.040,21.943,153.910
C08677=1074.006,-46.337,-58.990,173.038,21.941,153.910
C08678=1074.001,-46.586,-58.978,173.037,21.939,153.910
C08679=1073.995,-46.837,-58.967,173.035,21.937,153.910
C08680=1073.989,-47.087,-58.954,173.034,21.934,153.909
C08681=1073.983,-47.336,-58.942,173.033,21.932,153.909
C08682=1073.977,-47.585,-58.930,173.031,21.931,153.909
C08683=1073.971,-47.835,-58.917,173.030,21.929,153.909
C08684=1073.965,-48.085,-58.905,173.028,21.927,153.909
C08685=1073.959,-48.334,-58.893,173.027,21.925,153.909
C08686=1073.953,-48.584,-58.881,173.026,21.923,153.909
C08687=1073.946,-48.833,-58.869,173.024,21.921,153.908
C08688=1073.941,-49.083,-58.857,173.022,21.918,153.908
C08689=1073.934,-49.359,-58.843,173.021,21.916,153.908
C08690=1073.927,-49.635,-58.830,173.019,21.914,153.908
C08691=1073.921,-49.911,-58.816,173.018,21.912,153.908
C08692=1073.915,-50.187,-58.804,173.016,21.909,153.907
C08693=1073.908,-50.436,-58.792,173.015,21.907,153.907
C08694=1073.903,-50.686,-58.779,173.013,21.905,153.907
C08695=1073.896,-50.935,-58.767,173.012,21.903,153.907
C08696=1073.890,-51.185,-58.755,173.010,21.902,153.907
C08697=1073.884,-51.435,-58.744,173.009,21.900,153.907
C08698=1073.878,-51.684,-58.732,173.008,21.898,153.906
C08699=1073.872,-51.934,-58.719,173.006,21.896,153.906
C08700=1073.866,-52.184,-58.708,173.005,21.894,153.906
C08701=1073.859,-52.433,-58.696,173.002,21.892,153.906
C08702=1073.854,-52.683,-58.684,173.001,21.890,153.906
C08703=1073.847,-52.932,-58.672,173.000,21.888,153.906
C08704=1073.841,-53.182,-58.660,172.998,21.886,153.906
C08705=1073.835,-53.431,-58.648,172.997,21.884,153.906
C08706=1073.829,-53.681,-58.637,172.996,21.882,153.905
C08707=1073.822,-53.931,-58.625,172.994,21.880,153.905
C08708=1073.817,-54.180,-58.613,172.993,21.878,153.905
C08709=1073.811,-54.430,-58.601,172.991,21.877,153.905
C08710=1073.804,-54.680,-58.589,172.990,21.875,153.905
C08711=1073.798,-54.930,-58.577,172.988,21.873,153.905
C08712=1073.792,-55.179,-58.566,172.987,21.871,153.905
C08713=1073.786,-55.429,-58.554,172.985,21.869,153.905
C08714=1073.780,-55.679,-58.541,172.983,21.867,153.904
C08715=1073.774,-55.928,-58.531,172.982,21.865,153.904
C08716=1073.767,-56.178,-58.519,172.981,21.863,153.904
C08717=1073.761,-56.428,-58.506,172.979,21.861,153.904
C08718=1073.756,-56.677,-58.495,172.978,21.859,153.904
C08719=1073.749,-56.927,-58.483,172.976,21.858,153.904
C08720=1073.744,-57.176,-58.471,172.975,21.856,153.904
C08721=1073.737,-57.426,-58.460,172.974,21.854,153.903
C08722=1073.731,-57.676,-58.448,172.972,21.852,153.903
C08723=1073.725,-57.925,-58.437,172.971,21.850,153.903
C08724=1073.719,-58.175,-58.424,172.969,21.848,153.903
C08725=1073.713,-58.425,-58.412,172.968,21.846,153.903
C08726=1073.707,-58.674,-58.402,172.966,21.844,153.903
C08727=1073.701,-58.924,-58.389,172.964,21.843,153.903
C08728=1073.695,-59.174,-58.378,172.963,21.841,153.903
C08729=1073.688,-59.423,-58.366,172.961,21.839,153.902
C08730=1073.682,-59.673,-58.355,172.960,21.837,153.902
C08731=1073.677,-59.922,-58.343,172.959,21.835,153.902
C08732=1073.670,-60.173,-58.331,172.957,21.833,153.902
C08733=1073.664,-60.422,-58.320,172.956,21.831,153.902
C08734=1073.659,-60.671,-58.307,172.954,21.830,153.902
C08735=1073.653,-60.921,-58.296,172.953,21.828,153.902
C08736=1073.646,-61.170,-58.284,172.952,21.826,153.901
C08737=1073.640,-61.421,-58.273,172.950,21.824,153.901
C08738=1073.634,-61.670,-58.261,172.949,21.822,153.901
C08739=1073.628,-61.920,-58.250,172.947,21.820,153.901
C08740=1073.622,-62.170,-58.239,172.945,21.818,153.901
C08741=1073.616,-62.419,-58.227,172.944,21.816,153.901
C08742=1073.611,-62.669,-58.216,172.942,21.815,153.901
C08743=1073.604,-62.918,-58.204,172.941,21.813,153.901
C08744=1073.598,-63.168,-58.193,172.939,21.811,153.901
C08745=1073.592,-63.418,-58.181,172.938,21.809,153.900
C08746=1073.586,-63.667,-58.170,172.936,21.807,153.900
C08747=1073.580,-63.917,-58.157,172.935,21.806,153.900
C08748=1073.574,-64.167,-58.146,172.934,21.804,153.900
C08749=1073.568,-64.417,-58.135,172.932,21.802,153.900
C08750=1073.561,-64.666,-58.123,172.931,21.800,153.900
C08751=1073.556,-64.916,-58.112,172.929,21.798,153.900
C08752=1073.550,-65.166,-58.100,172.928,21.796,153.900
C08753=1073.544,-65.442,-58.088,172.926,21.794,153.899
C08754=1073.537,-65.719,-58.075,172.924,21.792,153.899
C08755=1073.530,-65.997,-58.063,172.923,21.790,153.899
C08756=1073.523,-66.273,-58.049,172.922,21.788,153.899
C08757=1073.517,-66.523,-58.039,172.920,21.787,153.899
C08758=1073.512,-66.773,-58.027,172.918,21.784,153.899
C08759=1073.506,-67.022,-58.015,172.916,21.783,153.899
C08760=1073.499,-67.273,-58.004,172.915,21.781,153.899
C08761=1073.494,-67.522,-57.993,172.913,21.779,153.899
C08762=1073.487,-67.772,-57.981,172.912,21.777,153.898
C08763=1073.482,-68.021,-57.970,172.911,21.775,153.898
C08764=1073.476,-68.272,-57.958,172.909,21.774,153.898
C08765=1073.470,-68.520,-57.947,172.908,21.772,153.898
C08766=1073.464,-68.770,-57.936,172.906,21.770,153.898
C08767=1073.457,-69.020,-57.925,172.905,21.769,153.898
C08768=1073.452,-69.270,-57.914,172.903,21.767,153.898
C08769=1073.446,-69.520,-57.901,172.902,21.765,153.898
C08770=1073.440,-69.769,-57.890,172.900,21.763,153.898
C08771=1073.434,-70.019,-57.879,172.899,21.761,153.897
C08772=1073.428,-70.269,-57.868,172.898,21.760,153.897
C08773=1073.422,-70.518,-57.857,172.896,21.758,153.897
C08774=1073.416,-70.768,-57.845,172.895,21.756,153.897
C08775=1073.411,-71.018,-57.834,172.893,21.754,153.897
C08776=1073.405,-71.267,-57.823,172.892,21.753,153.897
C08777=1073.398,-71.517,-57.811,172.890,21.750,153.897
C08778=1073.392,-71.766,-57.800,172.888,21.749,153.897
C08779=1073.386,-72.016,-57.789,172.887,21.747,153.897
C08780=1073.380,-72.266,-57.778,172.885,21.745,153.897
C08781=1073.375,-72.515,-57.767,172.884,21.743,153.896
C08782=1073.369,-72.766,-57.755,172.882,21.742,153.896
C08783=1073.363,-73.015,-57.744,172.881,21.740,153.896
C08784=1073.357,-73.264,-57.733,172.879,21.739,153.896
C08785=1073.351,-73.514,-57.722,172.878,21.737,153.896
C08786=1073.345,-73.764,-57.711,172.877,21.735,153.896
C08787=1073.339,-74.013,-57.700,172.875,21.733,153.896
C08788=1073.333,-74.263,-57.689,172.874,21.731,153.896
C08789=1073.327,-74.513,-57.678,172.872,21.730,153.896
C08790=1073.321,-74.763,-57.666,172.871,21.728,153.896
C08791=1073.315,-75.012,-57.655,172.869,21.727,153.896
C08792=1073.309,-75.262,-57.644,172.868,21.725,153.895
C08793=1073.303,-75.512,-57.633,172.866,21.723,153.895
C08794=1073.297,-75.761,-57.622,172.865,21.721,153.895
C08795=1073.290,-76.011,-57.611,172.863,21.720,153.895
C08796=1073.284,-76.261,-57.600,172.862,21.718,153.895
C08797=1073.279,-76.510,-57.590,172.860,21.717,153.895
C08798=1073.272,-76.760,-57.578,172.859,21.715,153.895
C08799=1073.267,-77.010,-57.567,172.857,21.713,153.895
C08800=1073.261,-77.259,-57.557,172.856,21.712,153.895
C08801=1073.254,-77.509,-57.545,172.854,21.710,153.895
C08802=1073.249,-77.759,-57.534,172.853,21.709,153.895
C08803=1073.242,-78.009,-57.523,172.851,21.706,153.895
C08804=1073.237,-78.259,-57.512,172.849,21.705,153.895
C08805=1073.230,-78.507,-57.501,172.847,21.703,153.894
C08806=1073.223,-78.757,-57.490,172.846,21.701,153.894
C08807=1073.218,-79.007,-57.479,172.844,21.700,153.894
C08808=1073.212,-79.257,-57.469,172.843,21.698,153.894
C08809=1073.207,-79.506,-57.458,172.842,21.697,153.894
C08810=1073.200,-79.757,-57.447,172.840,21.695,153.894
C08811=1073.194,-80.006,-57.436,172.839,21.693,153.894
C08812=1073.187,-80.256,-57.425,172.837,21.692,153.894
C08813=1073.182,-80.505,-57.414,172.835,21.691,153.894
C08814=1073.176,-80.755,-57.404,172.834,21.689,153.894
C08815=1073.169,-81.005,-57.393,172.832,21.687,153.894
C08816=1073.163,-81.254,-57.382,172.831,21.686,153.894
C08817=1073.156,-81.533,-57.370,172.830,21.684,153.894
C08818=1073.149,-81.813,-57.358,172.828,21.683,153.894
C08819=1073.142,-82.092,-57.345,172.826,21.681,153.894
C08820=1073.136,-82.371,-57.334,172.824,21.679,153.893
C08821=1073.129,-82.621,-57.323,172.823,21.677,153.893
C08822=1073.123,-82.871,-57.312,172.821,21.676,153.893
C08823=1073.117,-83.120,-57.302,172.820,21.674,153.893
C08824=1073.111,-83.370,-57.290,172.818,21.673,153.893
C08825=1073.104,-83.619,-57.280,172.817,21.671,153.893
C08826=1073.099,-83.870,-57.270,172.815,21.670,153.893
C08827=1073.093,-84.119,-57.259,172.813,21.668,153.893
C08828=1073.086,-84.369,-57.248,172.812,21.667,153.893
C08829=1073.080,-84.618,-57.238,172.810,21.665,153.893
C08830=1073.075,-84.868,-57.227,172.809,21.664,153.893
C08831=1073.068,-85.118,-57.216,172.807,21.662,153.893
C08832=1073.062,-85.368,-57.206,172.806,21.661,153.893
C08833=1073.056,-85.617,-57.195,172.804,21.659,153.893
C08834=1073.049,-85.867,-57.184,172.803,21.658,153.893
C08835=1073.044,-86.117,-57.173,172.801,21.656,153.893
C08836=1073.038,-86.366,-57.163,172.800,21.655,153.893
C08837=1073.032,-86.616,-57.153,172.798,21.653,153.893
C08838=1073.025,-86.866,-57.142,172.797,21.651,153.893
C08839=1073.020,-87.116,-57.131,172.795,21.650,153.893
C08840=1073.013,-87.365,-57.121,172.794,21.649,153.893
C08841=1073.008,-87.615,-57.110,172.792,21.647,153.893
C08842=1073.001,-87.865,-57.100,172.790,21.646,153.893
C08843=1072.995,-88.114,-57.089,172.789,21.645,153.893
C08844=1072.989,-88.364,-57.078,172.787,21.643,153.892
C08845=1072.983,-88.614,-57.068,172.786,21.641,153.892
C08846=1072.977,-88.864,-57.057,172.784,21.640,153.892
C08847=1072.970,-89.113,-57.047,172.783,21.638,153.892
C08848=1072.964,-89.363,-57.036,172.781,21.637,153.892
C08849=1072.959,-89.613,-57.026,172.780,21.636,153.892
C08850=1072.952,-89.862,-57.016,172.778,21.634,153.892
C08851=1072.946,-90.112,-57.004,172.777,21.633,153.892
C08852=1072.940,-90.362,-56.995,172.775,21.631,153.892
C08853=1072.934,-90.611,-56.984,172.773,21.630,153.892
C08854=1072.928,-90.861,-56.973,172.772,21.628,153.892
C08855=1072.922,-91.111,-56.963,172.770,21.627,153.892
C08856=1072.916,-91.361,-56.952,172.769,21.625,153.892
C08857=1072.909,-91.610,-56.942,172.767,21.624,153.892
C08858=1072.904,-91.860,-56.932,172.766,21.622,153.892
C08859=1072.898,-92.110,-56.921,172.764,21.621,153.892
C08860=1072.892,-92.359,-56.911,172.763,21.620,153.892
C08861=1072.886,-92.609,-56.900,172.761,21.618,153.892
C08862=1072.879,-92.859,-56.890,172.759,21.617,153.892
C08863=1072.874,-93.109,-56.880,172.758,21.616,153.892
C08864=1072.867,-93.358,-56.869,172.756,21.614,153.892
C08865=1072.862,-93.608,-56.859,172.755,21.613,153.892
C08866=1072.856,-93.858,-56.848,172.753,21.611,153.892
C08867=1072.850,-94.107,-56.838,172.752,21.610,153.892
C08868=1072.844,-94.357,-56.828,172.750,21.609,153.892
C08869=1072.837,-94.607,-56.817,172.748,21.607,153.892
C08870=1072.832,-94.857,-56.807,172.747,21.606,153.892
C08871=1072.825,-95.106,-56.797,172.745,21.604,153.892
C08872=1072.820,-95.356,-56.787,172.744,21.603,153.892
C08873=1072.813,-95.605,-56.776,172.742,21.602,153.892
C08874=1072.808,-95.855,-56.766,172.741,21.600,153.892
C08875=1072.801,-96.105,-56.756,172.739,21.599,153.892
C08876=1072.796,-96.355,-56.746,172.738,21.597,153.892
C08877=1072.790,-96.604,-56.735,172.736,21.596,153.892
C08878=1072.784,-96.853,-56.725,172.734,21.595,153.892
C08879=1072.777,-97.104,-56.715,172.733,21.593,153.892
C08880=1072.772,-97.354,-56.704,172.731,21.592,153.892
C08881=1072.765,-97.635,-56.693,172.730,21.590,153.892
C08882=1072.758,-97.916,-56.681,172.728,21.589,153.892
C08883=1072.751,-98.199,-56.670,172.727,21.588,153.892
C08884=1072.744,-98.480,-56.659,172.724,21.586,153.892
C08885=1072.738,-98.729,-56.648,172.723,21.584,153.892
C08886=1072.732,-98.979,-56.638,172.721,21.583,153.892
C08887=1072.725,-99.229,-56.629,172.719,21.582,153.892
C08888=1072.720,-99.479,-56.618,172.719,21.581,153.892
C08889=1072.714,-99.728,-56.608,172.717,21.580,153.892
C08890=1072.707,-99.977,-56.598,172.715,21.578,153.892
C08891=1072.702,-100.228,-56.588,172.714,21.577,153.892
C08892=1072.695,-100.477,-56.578,172.712,21.576,153.892
C08893=1072.688,-100.727,-56.567,172.710,21.575,153.892
C08894=1072.683,-100.977,-56.557,172.709,21.573,153.892
C08895=1072.676,-101.227,-56.547,172.707,21.572,153.892
C08896=1072.670,-101.476,-56.537,172.706,21.571,153.892
C08897=1072.665,-101.726,-56.527,172.704,21.570,153.892
C08898=1072.658,-101.976,-56.517,172.702,21.568,153.892
C08899=1072.652,-102.225,-56.507,172.701,21.567,153.892
C08900=1072.647,-102.476,-56.497,172.699,21.566,153.892
C08901=1072.640,-102.725,-56.487,172.698,21.565,153.892
C08902=1072.634,-102.975,-56.477,172.696,21.563,153.892
C08903=1072.628,-103.224,-56.468,172.694,21.562,153.892
C08904=1072.622,-103.474,-56.457,172.693,21.560,153.892
C08905=1072.616,-103.724,-56.447,172.691,21.560,153.892
C08906=1072.610,-103.973,-56.438,172.690,21.558,153.892
C08907=1072.603,-104.223,-56.428,172.688,21.557,153.892
C08908=1072.598,-104.473,-56.417,172.686,21.555,153.892
C08909=1072.592,-104.723,-56.408,172.685,21.555,153.892
C08910=1072.585,-104.972,-56.398,172.683,21.553,153.892
C08911=1072.579,-105.222,-56.387,172.681,21.552,153.892
C08912=1072.573,-105.472,-56.377,172.681,21.551,153.892
C08913=1072.567,-105.722,-56.368,172.679,21.550,153.892
C08914=1072.560,-105.971,-56.358,172.677,21.549,153.892
C08915=1072.554,-106.221,-56.348,172.676,21.548,153.892
C08916=1072.549,-106.471,-56.338,172.674,21.546,153.892
C08917=1072.543,-106.721,-56.328,172.673,21.545,153.892
C08918=1072.536,-106.970,-56.318,172.671,21.544,153.892
C08919=1072.530,-107.220,-56.308,172.669,21.543,153.892
C08920=1072.525,-107.470,-56.298,172.667,21.542,153.892
C08921=1072.518,-107.720,-56.289,172.666,21.540,153.892
C08922=1072.512,-107.970,-56.279,172.664,21.539,153.892
C08923=1072.506,-108.219,-56.269,172.663,21.538,153.892
C08924=1072.500,-108.469,-56.259,172.661,21.537,153.892
C08925=1072.493,-108.718,-56.250,172.659,21.536,153.892
C08926=1072.487,-108.968,-56.240,172.658,21.535,153.892
C08927=1072.481,-109.218,-56.231,172.656,21.534,153.892
C08928=1072.475,-109.468,-56.221,172.654,21.532,153.892
C08929=1072.469,-109.717,-56.210,172.653,21.532,153.893
C08930=1072.463,-109.967,-56.201,172.652,21.531,153.892
C08931=1072.457,-110.217,-56.191,172.650,21.530,153.893
C08932=1072.451,-110.467,-56.182,172.649,21.528,153.893
C08933=1072.445,-110.717,-56.172,172.647,21.527,153.893
C08934=1072.438,-110.966,-56.162,172.645,21.526,153.893
C08935=1072.432,-111.216,-56.153,172.643,21.525,153.893
C08936=1072.426,-111.466,-56.143,172.642,21.524,153.893
C08937=1072.420,-111.715,-56.134,172.640,21.523,153.893
C08938=1072.414,-111.964,-56.124,172.639,21.522,153.893
C08939=1072.408,-112.214,-56.114,172.637,21.521,153.893
C08940=1072.402,-112.464,-56.105,172.635,21.519,153.893
C08941=1072.396,-112.714,-56.094,172.633,21.518,153.893
C08942=1072.390,-112.964,-56.085,172.632,21.517,153.893
C08943=1072.384,-113.213,-56.075,172.630,21.516,153.893
C08944=1072.378,-113.463,-56.066,172.629,21.515,153.893
C08945=1072.370,-113.742,-56.055,172.627,21.514,153.893
C08946=1072.364,-114.021,-56.045,172.625,21.513,153.893
C08947=1072.357,-114.300,-56.034,172.623,21.512,153.893
C08948=1072.349,-114.579,-56.023,172.622,21.510,153.893
C08949=1072.343,-114.829,-56.013,172.620,21.510,153.894
C08950=1072.337,-115.079,-56.004,172.618,21.509,153.894
C08951=1072.332,-115.328,-55.995,172.617,21.507,153.894
C08952=1072.325,-115.578,-55.985,172.615,21.506,153.894
C08953=1072.319,-115.828,-55.975,172.613,21.506,153.894
C08954=1072.313,-116.077,-55.966,172.612,21.504,153.894
C08955=1072.307,-116.327,-55.956,172.611,21.504,153.894
C08956=1072.301,-116.578,-55.947,172.609,21.503,153.894
C08957=1072.295,-116.827,-55.938,172.607,21.502,153.894
C08958=1072.289,-117.077,-55.928,172.606,21.501,153.894
C08959=1072.282,-117.327,-55.919,172.604,21.500,153.894
C08960=1072.276,-117.577,-55.909,172.602,21.498,153.894
C08961=1072.270,-117.827,-55.900,172.601,21.498,153.894
C08962=1072.265,-118.076,-55.890,172.599,21.497,153.894
C08963=1072.258,-118.326,-55.881,172.597,21.495,153.894
C08964=1072.252,-118.575,-55.871,172.596,21.495,153.895
C08965=1072.246,-118.825,-55.862,172.594,21.494,153.895
C08966=1072.239,-119.075,-55.853,172.593,21.493,153.895
C08967=1072.233,-119.324,-55.843,172.591,21.492,153.895
C08968=1072.227,-119.574,-55.834,172.590,21.491,153.895
C08969=1072.221,-119.825,-55.825,172.588,21.490,153.895
C08970=1072.215,-120.074,-55.816,172.586,21.489,153.895
C08971=1072.209,-120.324,-55.806,172.584,21.488,153.895
C08972=1072.203,-120.573,-55.796,172.583,21.487,153.895
C08973=1072.197,-120.823,-55.787,172.581,21.486,153.895
C08974=1072.191,-121.073,-55.777,172.579,21.485,153.895
C08975=1072.184,-121.322,-55.768,172.578,21.485,153.895
C08976=1072.178,-121.573,-55.759,172.577,21.484,153.895
C08977=1072.172,-121.822,-55.750,172.575,21.483,153.896
C08978=1072.166,-122.072,-55.741,172.573,21.482,153.896
C08979=1072.160,-122.322,-55.731,172.571,21.481,153.896
C08980=1072.154,-122.571,-55.722,172.570,21.480,153.896
C08981=1072.148,-122.822,-55.713,172.568,21.479,153.896
C08982=1072.141,-123.071,-55.704,172.566,21.478,153.896
C08983=1072.135,-123.320,-55.695,172.565,21.477,153.896
C08984=1072.129,-123.570,-55.685,172.563,21.476,153.896
C08985=1072.123,-123.820,-55.675,172.562,21.476,153.896
C08986=1072.117,-124.070,-55.667,172.560,21.475,153.896
C08987=1072.110,-124.320,-55.658,172.558,21.474,153.897
C08988=1072.105,-124.569,-55.648,172.557,21.473,153.897
C08989=1072.099,-124.819,-55.639,172.555,21.472,153.897
C08990=1072.093,-125.069,-55.630,172.553,21.471,153.897
C08991=1072.086,-125.319,-55.621,172.551,21.470,153.897
C08992=1072.080,-125.568,-55.611,172.550,21.469,153.897
C08993=1072.073,-125.818,-55.602,172.549,21.469,153.897
C08994=1072.068,-126.068,-55.593,172.547,21.468,153.897
C08995=1072.061,-126.317,-55.584,172.545,21.467,153.897
C08996=1072.055,-126.567,-55.575,172.544,21.466,153.897
C08997=1072.049,-126.818,-55.566,172.542,21.466,153.898
C08998=1072.043,-127.067,-55.556,172.540,21.465,153.898
C08999=1072.037,-127.316,-55.548,172.538,21.464,153.898
C09000=1072.031,-127.567,-55.539,172.536,21.463,153.898
C09001=1072.024,-127.818,-55.530,172.536,21.463,153.898
C09002=1072.019,-128.068,-55.520,172.534,21.462,153.898
C09003=1072.016,-128.319,-55.509,172.532,21.460,153.898
C09004=1072.014,-128.569,-55.499,172.531,21.457,153.898
C09005=1072.015,-128.822,-55.487,172.530,21.454,153.897
C09006=1072.019,-129.075,-55.474,172.530,21.450,153.897
C09007=1072.024,-129.327,-55.460,172.529,21.445,153.896
C09008=1072.032,-129.577,-55.445,172.530,21.439,153.895
C09009=1071.641,-129.600,-55.607,172.483,21.576,153.927
C09010=1071.632,-129.349,-55.622,172.483,21.581,153.928
C09011=1071.627,-129.097,-55.636,172.484,21.586,153.928
C09012=1071.624,-128.844,-55.649,172.484,21.590,153.929
C09013=1071.623,-128.591,-55.661,172.485,21.594,153.930
C09014=1071.624,-128.341,-55.673,172.486,21.596,153.930
C09015=1071.627,-128.090,-55.683,172.487,21.598,153.930
C09016=1071.632,-127.839,-55.692,172.489,21.599,153.930
C09017=1071.638,-127.589,-55.701,172.491,21.600,153.930
C09018=1071.645,-127.339,-55.710,172.493,21.601,153.930
C09019=1071.651,-127.089,-55.719,172.495,21.602,153.930
C09020=1071.657,-126.839,-55.728,172.495,21.602,153.929
C09021=1071.663,-126.589,-55.738,172.497,21.603,153.929
C09022=1071.669,-126.340,-55.746,172.499,21.604,153.929
C09023=1071.675,-126.090,-55.755,172.501,21.605,153.929
C09024=1071.681,-125.840,-55.765,172.502,21.606,153.929
C09025=1071.688,-125.591,-55.774,172.504,21.607,153.929
C09026=1071.694,-125.341,-55.783,172.506,21.608,153.929
C09027=1071.700,-125.091,-55.792,172.508,21.608,153.929
C09028=1071.706,-124.842,-55.802,172.508,21.609,153.929
C09029=1071.713,-124.592,-55.811,172.510,21.610,153.929
C09030=1071.718,-124.342,-55.819,172.512,21.610,153.928
C09031=1071.725,-124.092,-55.829,172.514,21.611,153.928
C09032=1071.731,-123.842,-55.839,172.516,21.612,153.928
C09033=1071.736,-123.593,-55.848,172.517,21.613,153.928
C09034=1071.743,-123.343,-55.856,172.519,21.614,153.928
C09035=1071.749,-123.093,-55.866,172.521,21.615,153.928
C09036=1071.755,-122.843,-55.875,172.522,21.616,153.928
C09037=1071.762,-122.594,-55.885,172.523,21.616,153.928
C09038=1071.768,-122.344,-55.894,172.525,21.617,153.928
C09039=1071.773,-122.094,-55.903,172.527,21.618,153.928
C09040=1071.780,-121.845,-55.912,172.528,21.620,153.928
C09041=1071.786,-121.595,-55.921,172.530,21.620,153.928
C09042=1071.792,-121.345,-55.931,172.532,21.621,153.927
C09043=1071.798,-121.095,-55.940,172.534,21.622,153.927
C09044=1071.805,-120.845,-55.950,172.536,21.623,153.927
C09045=1071.810,-120.596,-55.959,172.537,21.624,153.927
C09046=1071.816,-120.346,-55.968,172.539,21.625,153.927
C09047=1071.822,-120.096,-55.978,172.540,21.626,153.927
C09048=1071.829,-119.847,-55.987,172.542,21.626,153.927
C09049=1071.835,-119.597,-55.996,172.543,21.628,153.927
C09050=1071.841,-119.347,-56.006,172.545,21.629,153.927
C09051=1071.848,-119.097,-56.015,172.547,21.629,153.927
C09052=1071.854,-118.847,-56.025,172.548,21.630,153.927
C09053=1071.859,-118.598,-56.033,172.550,21.632,153.927
C09054=1071.865,-118.348,-56.043,172.552,21.633,153.926
C09055=1071.871,-118.098,-56.053,172.554,21.633,153.926
C09056=1071.878,-117.848,-56.062,172.555,21.635,153.926
C09057=1071.884,-117.598,-56.072,172.557,21.636,153.926
C09058=1071.890,-117.349,-56.081,172.558,21.636,153.926
C09059=1071.897,-117.099,-56.090,172.560,21.637,153.926
C09060=1071.903,-116.849,-56.100,172.561,21.638,153.926
C09061=1071.909,-116.600,-56.109,172.563,21.639,153.926
C09062=1071.915,-116.350,-56.119,172.565,21.640,153.926
C09063=1071.921,-116.101,-56.128,172.566,21.641,153.926
C09064=1071.927,-115.851,-56.138,172.568,21.642,153.926
C09065=1071.933,-115.601,-56.147,172.570,21.644,153.926
C09066=1071.939,-115.351,-56.157,172.571,21.644,153.926
C09067=1071.946,-115.102,-56.166,172.573,21.645,153.926
C09068=1071.952,-114.852,-56.176,172.575,21.647,153.926
C09069=1071.958,-114.602,-56.186,172.576,21.647,153.925
C09070=1071.964,-114.322,-56.196,172.578,21.648,153.925
C09071=1071.971,-114.044,-56.207,172.580,21.650,153.925
C09072=1071.978,-113.764,-56.218,172.582,21.650,153.925
C09073=1071.985,-113.485,-56.228,172.583,21.652,153.925
C09074=1071.991,-113.235,-56.238,172.585,21.653,153.925
C09075=1071.997,-112.985,-56.247,172.586,21.654,153.925
C09076=1072.004,-112.735,-56.257,172.588,21.655,153.925
C09077=1072.010,-112.486,-56.266,172.590,21.656,153.925
C09078=1072.016,-112.236,-56.276,172.592,21.657,153.925
C09079=1072.022,-111.987,-56.286,172.593,21.659,153.925
C09080=1072.028,-111.737,-56.296,172.595,21.659,153.925
C09081=1072.034,-111.487,-56.306,172.596,21.661,153.925
C09082=1072.040,-111.237,-56.316,172.598,21.662,153.925
C09083=1072.046,-110.988,-56.325,172.599,21.663,153.925
C09084=1072.052,-110.738,-56.334,172.601,21.663,153.925
C09085=1072.058,-110.488,-56.344,172.602,21.665,153.925
C09086=1072.064,-110.239,-56.354,172.604,21.666,153.925
C09087=1072.070,-109.989,-56.363,172.606,21.667,153.925
C09088=1072.077,-109.740,-56.373,172.607,21.668,153.924
C09089=1072.083,-109.490,-56.383,172.609,21.669,153.924
C09090=1072.089,-109.240,-56.393,172.611,21.670,153.924
